LIN {X 0,Y 446.528,Z 466.485,A -85,B 0,C 180,E1 -8829.056,E2 -8829.056} C_VEL
LIN {X 0,Y 446.523,Z 466.485,A -85,B 0,C 180,E1 -8832.73,E2 -8832.73} C_VEL
LIN {X 0,Y 446.485,Z 466.496,A -85,B 0,C 180,E1 -8836.459,E2 -8836.459} C_VEL
LIN {X 0,Y 446.459,Z 466.494,A -85,B 0,C 180,E1 -8839.304,E2 -8839.304} C_VEL
LIN {X 0,Y 446.408,Z 466.501,A -85,B 0,C 180,E1 -8842.2,E2 -8842.2} C_VEL
LIN {X 0,Y 446.448,Z 466.494,A -85,B 0,C 180,E1 -8845.153,E2 -8845.153} C_VEL
LIN {X 0,Y 446.475,Z 466.494,A -85,B 0,C 180,E1 -8848.18,E2 -8848.18} C_VEL
LIN {X 0,Y 446.422,Z 466.498,A -85,B 0,C 180,E1 -8851.3,E2 -8851.3} C_VEL
LIN {X 0,Y 446.423,Z 466.501,A -85,B 0,C 180,E1 -8854.524,E2 -8854.524} C_VEL
LIN {X 0,Y 446.431,Z 466.498,A -85,B 0,C 180,E1 -8858.084,E2 -8858.084} C_VEL
LIN {X 0,Y 446.436,Z 466.501,A -85,B 0,C 180,E1 -8860.921,E2 -8860.921} C_VEL
LIN {X 0,Y 446.395,Z 466.503,A -85,B 0,C 180,E1 -8863.847,E2 -8863.847} C_VEL
LIN {X 0,Y 446.441,Z 466.501,A -85,B 0,C 180,E1 -8866.398,E2 -8866.398} C_VEL
LIN {X 0,Y 446.464,Z 466.495,A -85,B 0,C 180,E1 -8869.806,E2 -8869.806} C_VEL
LIN {X 0,Y 446.43,Z 466.501,A -85,B 0,C 180,E1 -8872.125,E2 -8872.125} C_VEL
LIN {X 0,Y 446.427,Z 466.499,A -85,B 0,C 180,E1 -8875.479,E2 -8875.479} C_VEL
LIN {X 0,Y 446.417,Z 466.5,A -85,B 0,C 180,E1 -8878.701,E2 -8878.701} C_VEL
LIN {X 0,Y 446.482,Z 466.498,A -85,B 0,C 180,E1 -8881.823,E2 -8881.823} C_VEL
LIN {X 0,Y 446.513,Z 466.543,A -85,B 0,C 180,E1 -8882.399,E2 -8882.399} C_VEL
LIN {X 0,Y 449.219,Z 479.048,A -85,B 0,C 180,E1 -8885.015,E2 -8885.015} C_VEL
LIN {X 0,Y 450.113,Z 484.167,A -85,B 0,C 180,E1 -8886.05,E2 -8886.05} C_VEL
LIN {X 0,Y 449.1,Z 500.867,A -85,B 0,C 180,E1 -8889.146,E2 -8889.146} C_VEL
LIN {X 0,Y 448.277,Z 515.978,A -85,B 0,C 180,E1 -8891.866,E2 -8891.866} C_VEL
LIN {X 0,Y 451.84,Z 534.729,A -85,B 0,C 180,E1 -8892.318,E2 -8892.318} C_VEL
LIN {X 0,Y 451.426,Z 605.013,A -85,B 0,C 180,E1 -8893.355,E2 -8893.355} C_VEL
LIN {X 0,Y 450.704,Z 610.873,A -85,B 0,C 180,E1 -8893.408,E2 -8893.408} C_VEL
LIN {X 0,Y 444.994,Z 629.85,A -85,B 0,C 180,E1 -8893.497,E2 -8893.497} C_VEL
LIN {X 0,Y 444.271,Z 635.605,A -85,B 0,C 180,E1 -8893.63,E2 -8893.63} C_VEL
LIN {X 0,Y 443.946,Z 647.952,A -85,B 0,C 180,E1 -8894.095,E2 -8894.095} C_VEL
LIN {X 0,Y 443.491,Z 657.945,A -85,B 0,C 180,E1 -8894.608,E2 -8894.608} C_VEL
LIN {X 0,Y 442.878,Z 668.385,A -85,B 0,C 180,E1 -8895.293,E2 -8895.293} C_VEL
LIN {X 0,Y 442.237,Z 679.403,A -85,B 0,C 180,E1 -8896.21,E2 -8896.21} C_VEL
LIN {X 0,Y 441.507,Z 688.316,A -85,B 0,C 180,E1 -8897.125,E2 -8897.125} C_VEL
LIN {X 0,Y 440.928,Z 697.479,A -85,B 0,C 180,E1 -8898.276,E2 -8898.276} C_VEL
LIN {X 0,Y 440.202,Z 706.324,A -85,B 0,C 180,E1 -8899.654,E2 -8899.654} C_VEL
LIN {X 0,Y 439.593,Z 713.46,A -85,B 0,C 180,E1 -8901.034,E2 -8901.034} C_VEL
LIN {X 0,Y 439.08,Z 720.054,A -85,B 0,C 180,E1 -8902.644,E2 -8902.644} C_VEL
LIN {X 0,Y 438.785,Z 724.416,A -85,B 0,C 180,E1 -8904.025,E2 -8904.025} C_VEL
LIN {X 0,Y 438.668,Z 727.741,A -85,B 0,C 180,E1 -8905.407,E2 -8905.407} C_VEL
LIN {X 0,Y 438.601,Z 729.446,A -85,B 0,C 180,E1 -8906.326,E2 -8906.326} C_VEL
LIN {X 0,Y 438.436,Z 731.666,A -85,B 0,C 180,E1 -8908.164,E2 -8908.164} C_VEL
LIN {X 0,Y 438.341,Z 732.451,A -85,B 0,C 180,E1 -8910.001,E2 -8910.001} C_VEL
LIN {X 0,Y 438.436,Z 731.738,A -85,B 0,C 180,E1 -8911.838,E2 -8911.838} C_VEL
LIN {X 0,Y 438.589,Z 729.577,A -85,B 0,C 180,E1 -8913.676,E2 -8913.676} C_VEL
LIN {X 0,Y 438.611,Z 726.93,A -85,B 0,C 180,E1 -8915.057,E2 -8915.057} C_VEL
LIN {X 0,Y 438.945,Z 723.319,A -85,B 0,C 180,E1 -8916.436,E2 -8916.436} C_VEL
LIN {X 0,Y 439.215,Z 718.662,A -85,B 0,C 180,E1 -8917.818,E2 -8917.818} C_VEL
LIN {X 0,Y 439.685,Z 712.8,A -85,B 0,C 180,E1 -8919.199,E2 -8919.199} C_VEL
LIN {X 0,Y 440.228,Z 705.527,A -85,B 0,C 180,E1 -8920.58,E2 -8920.58} C_VEL
LIN {X 0,Y 440.799,Z 698.102,A -85,B 0,C 180,E1 -8921.73,E2 -8921.73} C_VEL
LIN {X 0,Y 441.496,Z 689.112,A -85,B 0,C 180,E1 -8922.878,E2 -8922.878} C_VEL
LIN {X 0,Y 442.302,Z 678.809,A -85,B 0,C 180,E1 -8923.935,E2 -8923.935} C_VEL
LIN {X 0,Y 442.898,Z 668.024,A -85,B 0,C 180,E1 -8924.827,E2 -8924.827} C_VEL
LIN {X 0,Y 443.612,Z 655.51,A -85,B 0,C 180,E1 -8925.625,E2 -8925.625} C_VEL
LIN {X 0,Y 444.08,Z 643.304,A -85,B 0,C 180,E1 -8926.198,E2 -8926.198} C_VEL
LIN {X 0,Y 444.444,Z 630.676,A -85,B 0,C 180,E1 -8926.597,E2 -8926.597} C_VEL
LIN {X 0,Y 444.648,Z 612.531,A -85,B 0,C 180,E1 -8926.914,E2 -8926.914} C_VEL
LIN {X 0,Y 445.096,Z 535.017,A -85,B 0,C 180,E1 -8928.073,E2 -8928.073} C_VEL
LIN {X 0,Y 441.416,Z 515.921,A -85,B 0,C 180,E1 -8928.569,E2 -8928.569} C_VEL
LIN {X 0,Y 442.438,Z 498.957,A -85,B 0,C 180,E1 -8931.675,E2 -8931.675} C_VEL
LIN {X 0,Y 443.258,Z 486.092,A -85,B 0,C 180,E1 -8934.098,E2 -8934.098} C_VEL
LIN {X 0,Y 441.633,Z 477.096,A -85,B 0,C 180,E1 -8935.954,E2 -8935.954} C_VEL
LIN {X 0,Y 439.465,Z 467.377,A -85,B 0,C 180,E1 -8938.046,E2 -8938.046} C_VEL
LIN {X 0,Y 439.367,Z 467.386,A -85,B 0,C 180,E1 -8940.789,E2 -8940.789} C_VEL
LIN {X 0,Y 439.393,Z 467.377,A -85,B 0,C 180,E1 -8944.044,E2 -8944.044} C_VEL
LIN {X 0,Y 439.366,Z 467.383,A -85,B 0,C 180,E1 -8947.435,E2 -8947.435} C_VEL
LIN {X 0,Y 439.42,Z 467.377,A -85,B 0,C 180,E1 -8949.851,E2 -8949.851} C_VEL
LIN {X 0,Y 439.392,Z 467.376,A -85,B 0,C 180,E1 -8952.628,E2 -8952.628} C_VEL
LIN {X 0,Y 439.408,Z 467.372,A -85,B 0,C 180,E1 -8955.271,E2 -8955.271} C_VEL
LIN {X 0,Y 439.394,Z 467.372,A -85,B 0,C 180,E1 -8958.744,E2 -8958.744} C_VEL
LIN {X 0,Y 439.386,Z 467.374,A -85,B 0,C 180,E1 -8961.607,E2 -8961.607} C_VEL
LIN {X 0,Y 439.407,Z 467.372,A -85,B 0,C 180,E1 -8964.844,E2 -8964.844} C_VEL
LIN {X 0,Y 439.379,Z 467.379,A -85,B 0,C 180,E1 -8968.14,E2 -8968.14} C_VEL
LIN {X 0,Y 439.439,Z 467.373,A -85,B 0,C 180,E1 -8971.598,E2 -8971.598} C_VEL
LIN {X 0,Y 439.469,Z 467.447,A -85,B 0,C 180,E1 -8972.222,E2 -8972.222} C_VEL
LIN {X 0,Y 442.662,Z 482.424,A -85,B 0,C 180,E1 -8974.821,E2 -8974.821} C_VEL
LIN {X 0,Y 442.958,Z 486.098,A -85,B 0,C 180,E1 -8975.424,E2 -8975.424} C_VEL
LIN {X 0,Y 442.188,Z 505.789,A -85,B 0,C 180,E1 -8978.558,E2 -8978.558} C_VEL
LIN {X 0,Y 441.378,Z 528.036,A -85,B 0,C 180,E1 -8982.091,E2 -8982.091} C_VEL
LIN {X 0,Y 443.918,Z 544.485,A -85,B 0,C 180,E1 -8982.514,E2 -8982.514} C_VEL
LIN {X 0,Y 442.535,Z 638.568,A -85,B 0,C 180,E1 -8984.278,E2 -8984.278} C_VEL
LIN {X 0,Y 442.265,Z 651.117,A -85,B 0,C 180,E1 -8984.681,E2 -8984.681} C_VEL
LIN {X 0,Y 441.802,Z 664.471,A -85,B 0,C 180,E1 -8985.313,E2 -8985.313} C_VEL
LIN {X 0,Y 441.347,Z 676.321,A -85,B 0,C 180,E1 -8986.063,E2 -8986.063} C_VEL
LIN {X 0,Y 440.881,Z 687.275,A -85,B 0,C 180,E1 -8986.953,E2 -8986.953} C_VEL
LIN {X 0,Y 440.293,Z 697.9,A -85,B 0,C 180,E1 -8988.024,E2 -8988.024} C_VEL
LIN {X 0,Y 439.833,Z 707.197,A -85,B 0,C 180,E1 -8989.178,E2 -8989.178} C_VEL
LIN {X 0,Y 439.374,Z 716.17,A -85,B 0,C 180,E1 -8990.563,E2 -8990.563} C_VEL
LIN {X 0,Y 438.988,Z 723.4,A -85,B 0,C 180,E1 -8991.947,E2 -8991.947} C_VEL
LIN {X 0,Y 438.731,Z 729.051,A -85,B 0,C 180,E1 -8993.307,E2 -8993.307} C_VEL
LIN {X 0,Y 438.605,Z 732.967,A -85,B 0,C 180,E1 -8994.483,E2 -8994.483} C_VEL
LIN {X 0,Y 438.485,Z 736.528,A -85,B 0,C 180,E1 -8995.864,E2 -8995.864} C_VEL
LIN {X 0,Y 438.428,Z 739.05,A -85,B 0,C 180,E1 -8997.243,E2 -8997.243} C_VEL
LIN {X 0,Y 438.35,Z 740.174,A -85,B 0,C 180,E1 -8998.162,E2 -8998.162} C_VEL
LIN {X 0,Y 438.309,Z 740.884,A -85,B 0,C 180,E1 -8999.081,E2 -8999.081} C_VEL
LIN {X 0,Y 438.309,Z 741.198,A -85,B 0,C 180,E1 -9000,E2 -9000} C_VEL
LIN {X 0,Y 438.338,Z 741.073,A -85,B 0,C 180,E1 -9000.919,E2 -9000.919} C_VEL
LIN {X 0,Y 438.374,Z 740.513,A -85,B 0,C 180,E1 -9001.837,E2 -9001.837} C_VEL
LIN {X 0,Y 438.437,Z 739.553,A -85,B 0,C 180,E1 -9002.756,E2 -9002.756} C_VEL
LIN {X 0,Y 438.539,Z 738.167,A -85,B 0,C 180,E1 -9003.675,E2 -9003.675} C_VEL
LIN {X 0,Y 438.517,Z 735.243,A -85,B 0,C 180,E1 -9005.057,E2 -9005.057} C_VEL
LIN {X 0,Y 438.849,Z 731.225,A -85,B 0,C 180,E1 -9006.436,E2 -9006.436} C_VEL
LIN {X 0,Y 439.052,Z 725.028,A -85,B 0,C 180,E1 -9008.051,E2 -9008.051} C_VEL
LIN {X 0,Y 439.494,Z 718.222,A -85,B 0,C 180,E1 -9009.434,E2 -9009.434} C_VEL
LIN {X 0,Y 439.938,Z 709.665,A -85,B 0,C 180,E1 -9010.819,E2 -9010.819} C_VEL
LIN {X 0,Y 440.406,Z 700.881,A -85,B 0,C 180,E1 -9011.973,E2 -9011.973} C_VEL
LIN {X 0,Y 441.01,Z 690.712,A -85,B 0,C 180,E1 -9013.057,E2 -9013.057} C_VEL
LIN {X 0,Y 441.586,Z 679.066,A -85,B 0,C 180,E1 -9014.046,E2 -9014.046} C_VEL
LIN {X 0,Y 442.042,Z 666.93,A -85,B 0,C 180,E1 -9014.855,E2 -9014.855} C_VEL
LIN {X 0,Y 442.577,Z 654.201,A -85,B 0,C 180,E1 -9015.484,E2 -9015.484} C_VEL
LIN {X 0,Y 442.922,Z 642.024,A -85,B 0,C 180,E1 -9015.915,E2 -9015.915} C_VEL
LIN {X 0,Y 443.322,Z 620.082,A -85,B 0,C 180,E1 -9016.373,E2 -9016.373} C_VEL
LIN {X 0,Y 444.614,Z 543.316,A -85,B 0,C 180,E1 -9017.924,E2 -9017.924} C_VEL
LIN {X 0,Y 442.206,Z 530.197,A -85,B 0,C 180,E1 -9018.355,E2 -9018.355} C_VEL
LIN {X 0,Y 442.954,Z 509.029,A -85,B 0,C 180,E1 -9021.647,E2 -9021.647} C_VEL
LIN {X 0,Y 443.703,Z 490.09,A -85,B 0,C 180,E1 -9024.569,E2 -9024.569} C_VEL
LIN {X 0,Y 443.55,Z 484.614,A -85,B 0,C 180,E1 -9025.422,E2 -9025.422} C_VEL
LIN {X 0,Y 441.677,Z 475.467,A -85,B 0,C 180,E1 -9026.99,E2 -9026.99} C_VEL
LIN {X 0,Y 439.434,Z 467.377,A -85,B 0,C 180,E1 -9028.442,E2 -9028.442} C_VEL
LIN {X 0,Y 439.375,Z 467.384,A -85,B 0,C 180,E1 -9032.03,E2 -9032.03} C_VEL
LIN {X 0,Y 439.401,Z 467.377,A -85,B 0,C 180,E1 -9035.34,E2 -9035.34} C_VEL
LIN {X 0,Y 439.395,Z 467.376,A -85,B 0,C 180,E1 -9038.594,E2 -9038.594} C_VEL
LIN {X 0,Y 439.393,Z 467.378,A -85,B 0,C 180,E1 -9041.256,E2 -9041.256} C_VEL
LIN {X 0,Y 439.404,Z 467.375,A -85,B 0,C 180,E1 -9044.729,E2 -9044.729} C_VEL
LIN {X 0,Y 439.4,Z 467.378,A -85,B 0,C 180,E1 -9047.795,E2 -9047.795} C_VEL
LIN {X 0,Y 439.399,Z 467.374,A -85,B 0,C 180,E1 -9050.223,E2 -9050.223} C_VEL
LIN {X 0,Y 439.378,Z 467.38,A -85,B 0,C 180,E1 -9053.712,E2 -9053.712} C_VEL
LIN {X 0,Y 439.377,Z 467.381,A -85,B 0,C 180,E1 -9057.053,E2 -9057.053} C_VEL
LIN {X 0,Y 439.4,Z 467.425,A -85,B 0,C 180,E1 -9059.823,E2 -9059.823} C_VEL
LIN {X 0,Y 443.454,Z 483.224,A -85,B 0,C 180,E1 -9062.561,E2 -9062.561} C_VEL
LIN {X 0,Y 445.005,Z 490.464,A -85,B 0,C 180,E1 -9063.754,E2 -9063.754} C_VEL
LIN {X 0,Y 443.575,Z 510.491,A -85,B 0,C 180,E1 -9066.664,E2 -9066.664} C_VEL
LIN {X 0,Y 442.748,Z 522.844,A -85,B 0,C 180,E1 -9068.447,E2 -9068.447} C_VEL
LIN {X 0,Y 445.963,Z 544.781,A -85,B 0,C 180,E1 -9068.984,E2 -9068.984} C_VEL
LIN {X 0,Y 444.312,Z 657.862,A -85,B 0,C 180,E1 -9070.958,E2 -9070.958} C_VEL
LIN {X 0,Y 443.803,Z 672.315,A -85,B 0,C 180,E1 -9071.385,E2 -9071.385} C_VEL
LIN {X 0,Y 443.198,Z 685.875,A -85,B 0,C 180,E1 -9071.966,E2 -9071.966} C_VEL
LIN {X 0,Y 442.454,Z 700.183,A -85,B 0,C 180,E1 -9072.791,E2 -9072.791} C_VEL
LIN {X 0,Y 441.713,Z 712.707,A -85,B 0,C 180,E1 -9073.713,E2 -9073.713} C_VEL
LIN {X 0,Y 440.951,Z 724.181,A -85,B 0,C 180,E1 -9074.752,E2 -9074.752} C_VEL
LIN {X 0,Y 440.283,Z 734.747,A -85,B 0,C 180,E1 -9075.91,E2 -9075.91} C_VEL
LIN {X 0,Y 439.755,Z 744.042,A -85,B 0,C 180,E1 -9077.13,E2 -9077.13} C_VEL
LIN {X 0,Y 439.299,Z 752.571,A -85,B 0,C 180,E1 -9078.463,E2 -9078.463} C_VEL
LIN {X 0,Y 438.854,Z 761.143,A -85,B 0,C 180,E1 -9080.086,E2 -9080.086} C_VEL
LIN {X 0,Y 438.578,Z 768.005,A -85,B 0,C 180,E1 -9081.707,E2 -9081.707} C_VEL
LIN {X 0,Y 438.46,Z 772.747,A -85,B 0,C 180,E1 -9083.094,E2 -9083.094} C_VEL
LIN {X 0,Y 438.417,Z 777.575,A -85,B 0,C 180,E1 -9084.941,E2 -9084.941} C_VEL
LIN {X 0,Y 438.347,Z 780.144,A -85,B 0,C 180,E1 -9086.322,E2 -9086.322} C_VEL
LIN {X 0,Y 438.407,Z 781.414,A -85,B 0,C 180,E1 -9087.242,E2 -9087.242} C_VEL
LIN {X 0,Y 438.364,Z 782.86,A -85,B 0,C 180,E1 -9089.08,E2 -9089.08} C_VEL
LIN {X 0,Y 438.363,Z 782.861,A -85,B 0,C 180,E1 -9090.917,E2 -9090.917} C_VEL
LIN {X 0,Y 438.406,Z 781.418,A -85,B 0,C 180,E1 -9092.755,E2 -9092.755} C_VEL
LIN {X 0,Y 438.35,Z 778.515,A -85,B 0,C 180,E1 -9094.597,E2 -9094.597} C_VEL
LIN {X 0,Y 438.442,Z 774.291,A -85,B 0,C 180,E1 -9096.369,E2 -9096.369} C_VEL
LIN {X 0,Y 438.502,Z 769.686,A -85,B 0,C 180,E1 -9097.829,E2 -9097.829} C_VEL
LIN {X 0,Y 438.776,Z 763.241,A -85,B 0,C 180,E1 -9099.448,E2 -9099.448} C_VEL
LIN {X 0,Y 439.159,Z 755.192,A -85,B 0,C 180,E1 -9101.071,E2 -9101.071} C_VEL
LIN {X 0,Y 439.54,Z 747.348,A -85,B 0,C 180,E1 -9102.376,E2 -9102.376} C_VEL
LIN {X 0,Y 440.193,Z 736.626,A -85,B 0,C 180,E1 -9103.855,E2 -9103.855} C_VEL
LIN {X 0,Y 440.921,Z 725.347,A -85,B 0,C 180,E1 -9105.128,E2 -9105.128} C_VEL
LIN {X 0,Y 441.654,Z 714.136,A -85,B 0,C 180,E1 -9106.168,E2 -9106.168} C_VEL
LIN {X 0,Y 442.323,Z 701.958,A -85,B 0,C 180,E1 -9107.093,E2 -9107.093} C_VEL
LIN {X 0,Y 443.048,Z 689.083,A -85,B 0,C 180,E1 -9107.867,E2 -9107.867} C_VEL
LIN {X 0,Y 443.667,Z 675.303,A -85,B 0,C 180,E1 -9108.499,E2 -9108.499} C_VEL
LIN {X 0,Y 444.218,Z 661.187,A -85,B 0,C 180,E1 -9108.954,E2 -9108.954} C_VEL
LIN {X 0,Y 444.603,Z 640.583,A -85,B 0,C 180,E1 -9109.356,E2 -9109.356} C_VEL
LIN {X 0,Y 445.85,Z 543.854,A -85,B 0,C 180,E1 -9111.033,E2 -9111.033} C_VEL
LIN {X 0,Y 442.72,Z 522.592,A -85,B 0,C 180,E1 -9111.566,E2 -9111.566} C_VEL
LIN {X 0,Y 444.176,Z 502.158,A -85,B 0,C 180,E1 -9114.539,E2 -9114.539} C_VEL
LIN {X 0,Y 444.99,Z 490.428,A -85,B 0,C 180,E1 -9116.244,E2 -9116.244} C_VEL
LIN {X 0,Y 441.733,Z 476.236,A -85,B 0,C 180,E1 -9118.621,E2 -9118.621} C_VEL
LIN {X 0,Y 439.4,Z 467.374,A -85,B 0,C 180,E1 -9120.177,E2 -9120.177} C_VEL
LIN {X 0,Y 439.391,Z 467.374,A -85,B 0,C 180,E1 -9123.723,E2 -9123.723} C_VEL
LIN {X 0,Y 439.353,Z 467.384,A -85,B 0,C 180,E1 -9126.888,E2 -9126.888} C_VEL
LIN {X 0,Y 439.422,Z 467.372,A -85,B 0,C 180,E1 -9129.852,E2 -9129.852} C_VEL
LIN {X 0,Y 439.396,Z 467.379,A -85,B 0,C 180,E1 -9132.629,E2 -9132.629} C_VEL
LIN {X 0,Y 439.395,Z 467.373,A -85,B 0,C 180,E1 -9136.032,E2 -9136.032} C_VEL
LIN {X 0,Y 439.392,Z 467.375,A -85,B 0,C 180,E1 -9139.021,E2 -9139.021} C_VEL
LIN {X 0,Y 439.384,Z 467.372,A -85,B 0,C 180,E1 -9141.604,E2 -9141.604} C_VEL
LIN {X 0,Y 439.391,Z 467.365,A -85,B 0,C 180,E1 -9144.843,E2 -9144.843} C_VEL
LIN {X 0,Y 439.378,Z 467.376,A -85,B 0,C 180,E1 -9148.14,E2 -9148.14} C_VEL
LIN {X 0,Y 439.415,Z 467.37,A -85,B 0,C 180,E1 -9151.326,E2 -9151.326} C_VEL
LIN {X 0,Y 439.395,Z 467.379,A -85,B 0,C 180,E1 -9154.415,E2 -9154.415} C_VEL
LIN {X 0,Y 439.354,Z 467.361,A -85,B 0,C 180,E1 -9157.424,E2 -9157.424} C_VEL
LIN {X 0,Y 439.43,Z 467.37,A -85,B 0,C 180,E1 -9160.662,E2 -9160.662} C_VEL
LIN {X 0,Y 439.451,Z 467.366,A -85,B 0,C 180,E1 -9164.224,E2 -9164.224} C_VEL
LIN {X 0,Y 439.501,Z 467.36,A -85,B 0,C 180,E1 -9168.002,E2 -9168.002} C_VEL
LIN {X 0,Y 439.536,Z 467.356,A -85,B 0,C 180,E1 -9171.726,E2 -9171.726} C_VEL
LIN {X 0,Y 439.614,Z 467.346,A -85,B 0,C 180,E1 -9174.496,E2 -9174.496} C_VEL
LIN {X 0,Y 439.626,Z 467.345,A -85,B 0,C 180,E1 -9178.168,E2 -9178.168} C_VEL
LIN {X 0,Y 439.754,Z 467.328,A -85,B 0,C 180,E1 -9180,E2 -9180} C_VEL
LIN {X 0,Y 439.646,Z 467.34,A -85,B 0,C 180,E1 -9182.749,E2 -9182.749} C_VEL
LIN {X 0,Y 439.607,Z 467.353,A -85,B 0,C 180,E1 -9186.426,E2 -9186.426} C_VEL
LIN {X 0,Y 439.491,Z 467.36,A -85,B 0,C 180,E1 -9189.202,E2 -9189.202} C_VEL
LIN {X 0,Y 439.493,Z 467.36,A -85,B 0,C 180,E1 -9192.727,E2 -9192.727} C_VEL
LIN {X 0,Y 439.449,Z 467.372,A -85,B 0,C 180,E1 -9196.355,E2 -9196.355} C_VEL
LIN {X 0,Y 439.392,Z 467.374,A -85,B 0,C 180,E1 -9199.627,E2 -9199.627} C_VEL
LIN {X 0,Y 439.355,Z 467.38,A -85,B 0,C 180,E1 -9202.576,E2 -9202.576} C_VEL
LIN {X 0,Y 439.395,Z 467.372,A -85,B 0,C 180,E1 -9205.586,E2 -9205.586} C_VEL
LIN {X 0,Y 439.416,Z 467.375,A -85,B 0,C 180,E1 -9208.674,E2 -9208.674} C_VEL
LIN {X 0,Y 439.376,Z 467.378,A -85,B 0,C 180,E1 -9212.035,E2 -9212.035} C_VEL
LIN {X 0,Y 439.388,Z 467.375,A -85,B 0,C 180,E1 -9215.342,E2 -9215.342} C_VEL
LIN {X 0,Y 439.392,Z 467.381,A -85,B 0,C 180,E1 -9218.594,E2 -9218.594} C_VEL
LIN {X 0,Y 439.391,Z 467.376,A -85,B 0,C 180,E1 -9221.26,E2 -9221.26} C_VEL
LIN {X 0,Y 439.396,Z 467.378,A -85,B 0,C 180,E1 -9224.73,E2 -9224.73} C_VEL
LIN {X 0,Y 439.407,Z 467.374,A -85,B 0,C 180,E1 -9227.799,E2 -9227.799} C_VEL
LIN {X 0,Y 439.447,Z 467.371,A -85,B 0,C 180,E1 -9230.232,E2 -9230.232} C_VEL
LIN {X 0,Y 439.373,Z 467.374,A -85,B 0,C 180,E1 -9233.715,E2 -9233.715} C_VEL
LIN {X 0,Y 439.372,Z 467.381,A -85,B 0,C 180,E1 -9237.056,E2 -9237.056} C_VEL
LIN {X 0,Y 439.394,Z 467.378,A -85,B 0,C 180,E1 -9240.277,E2 -9240.277} C_VEL
LIN {X 0,Y 439.47,Z 467.469,A -85,B 0,C 180,E1 -9242.075,E2 -9242.075} C_VEL
LIN {X 0,Y 442.059,Z 479.194,A -85,B 0,C 180,E1 -9244.581,E2 -9244.581} C_VEL
LIN {X 0,Y 443.239,Z 485.599,A -85,B 0,C 180,E1 -9245.904,E2 -9245.904} C_VEL
LIN {X 0,Y 442.203,Z 502.354,A -85,B 0,C 180,E1 -9249.049,E2 -9249.049} C_VEL
LIN {X 0,Y 441.418,Z 515.939,A -85,B 0,C 180,E1 -9251.529,E2 -9251.529} C_VEL
LIN {X 0,Y 445.158,Z 535.672,A -85,B 0,C 180,E1 -9252.031,E2 -9252.031} C_VEL
LIN {X 0,Y 444.466,Z 628.207,A -85,B 0,C 180,E1 -9253.436,E2 -9253.436} C_VEL
LIN {X 0,Y 444.271,Z 635.605,A -85,B 0,C 180,E1 -9253.63,E2 -9253.63} C_VEL
LIN {X 0,Y 443.847,Z 639.428,A -85,B 0,C 180,E1 -9253.738,E2 -9253.738} C_VEL
LIN {X 0,Y 441.761,Z 646.881,A -85,B 0,C 180,E1 -9253.951,E2 -9253.951} C_VEL
LIN {X 0,Y 437.525,Z 658.588,A -85,B 0,C 180,E1 -9254.396,E2 -9254.396} C_VEL
LIN {X 0,Y 436.357,Z 664.758,A -85,B 0,C 180,E1 -9254.754,E2 -9254.754} C_VEL
LIN {X 0,Y 435.632,Z 676.154,A -85,B 0,C 180,E1 -9255.64,E2 -9255.64} C_VEL
LIN {X 0,Y 434.826,Z 686.741,A -85,B 0,C 180,E1 -9256.685,E2 -9256.685} C_VEL
LIN {X 0,Y 434.119,Z 696.253,A -85,B 0,C 180,E1 -9257.852,E2 -9257.852} C_VEL
LIN {X 0,Y 433.437,Z 704.057,A -85,B 0,C 180,E1 -9259.018,E2 -9259.018} C_VEL
LIN {X 0,Y 432.835,Z 711.727,A -85,B 0,C 180,E1 -9260.421,E2 -9260.421} C_VEL
LIN {X 0,Y 432.35,Z 716.928,A -85,B 0,C 180,E1 -9261.589,E2 -9261.589} C_VEL
LIN {X 0,Y 431.954,Z 721.974,A -85,B 0,C 180,E1 -9262.974,E2 -9262.974} C_VEL
LIN {X 0,Y 431.603,Z 726.039,A -85,B 0,C 180,E1 -9264.394,E2 -9264.394} C_VEL
LIN {X 0,Y 431.587,Z 728.162,A -85,B 0,C 180,E1 -9265.331,E2 -9265.331} C_VEL
LIN {X 0,Y 431.544,Z 729.86,A -85,B 0,C 180,E1 -9266.266,E2 -9266.266} C_VEL
LIN {X 0,Y 431.353,Z 732.076,A -85,B 0,C 180,E1 -9268.134,E2 -9268.134} C_VEL
LIN {X 0,Y 431.281,Z 732.859,A -85,B 0,C 180,E1 -9270.001,E2 -9270.001} C_VEL
LIN {X 0,Y 431.353,Z 732.148,A -85,B 0,C 180,E1 -9271.869,E2 -9271.869} C_VEL
LIN {X 0,Y 431.533,Z 729.989,A -85,B 0,C 180,E1 -9273.736,E2 -9273.736} C_VEL
LIN {X 0,Y 431.539,Z 727.349,A -85,B 0,C 180,E1 -9275.14,E2 -9275.14} C_VEL
LIN {X 0,Y 431.91,Z 723.744,A -85,B 0,C 180,E1 -9276.542,E2 -9276.542} C_VEL
LIN {X 0,Y 432.181,Z 719.097,A -85,B 0,C 180,E1 -9277.946,E2 -9277.946} C_VEL
LIN {X 0,Y 432.699,Z 713.245,A -85,B 0,C 180,E1 -9279.349,E2 -9279.349} C_VEL
LIN {X 0,Y 433.282,Z 705.984,A -85,B 0,C 180,E1 -9280.752,E2 -9280.752} C_VEL
LIN {X 0,Y 433.872,Z 698.578,A -85,B 0,C 180,E1 -9281.92,E2 -9281.92} C_VEL
LIN {X 0,Y 434.614,Z 689.615,A -85,B 0,C 180,E1 -9283.086,E2 -9283.086} C_VEL
LIN {X 0,Y 435.432,Z 679.539,A -85,B 0,C 180,E1 -9284.142,E2 -9284.142} C_VEL
LIN {X 0,Y 436.068,Z 668.622,A -85,B 0,C 180,E1 -9285.064,E2 -9285.064} C_VEL
LIN {X 0,Y 436.806,Z 656.18,A -85,B 0,C 180,E1 -9285.875,E2 -9285.875} C_VEL
LIN {X 0,Y 437.336,Z 643.401,A -85,B 0,C 180,E1 -9286.484,E2 -9286.484} C_VEL
LIN {X 0,Y 437.737,Z 630.664,A -85,B 0,C 180,E1 -9286.889,E2 -9286.889} C_VEL
LIN {X 0,Y 437.945,Z 612.328,A -85,B 0,C 180,E1 -9287.211,E2 -9287.211} C_VEL
LIN {X 0,Y 438.491,Z 536.306,A -85,B 0,C 180,E1 -9288.362,E2 -9288.362} C_VEL
LIN {X 0,Y 434.59,Z 515.966,A -85,B 0,C 180,E1 -9288.902,E2 -9288.902} C_VEL
LIN {X 0,Y 435.698,Z 497.838,A -85,B 0,C 180,E1 -9292.277,E2 -9292.277} C_VEL
LIN {X 0,Y 436.402,Z 487.52,A -85,B 0,C 180,E1 -9294.248,E2 -9294.248} C_VEL
LIN {X 0,Y 434.447,Z 477.241,A -85,B 0,C 180,E1 -9296.416,E2 -9296.416} C_VEL
LIN {X 0,Y 432.401,Z 468.255,A -85,B 0,C 180,E1 -9298.426,E2 -9298.426} C_VEL
LIN {X 0,Y 432.327,Z 468.262,A -85,B 0,C 180,E1 -9301.347,E2 -9301.347} C_VEL
LIN {X 0,Y 432.346,Z 468.253,A -85,B 0,C 180,E1 -9304.678,E2 -9304.678} C_VEL
LIN {X 0,Y 432.353,Z 468.251,A -85,B 0,C 180,E1 -9308.149,E2 -9308.149} C_VEL
LIN {X 0,Y 432.341,Z 468.255,A -85,B 0,C 180,E1 -9311.603,E2 -9311.603} C_VEL
LIN {X 0,Y 432.347,Z 468.25,A -85,B 0,C 180,E1 -9314.347,E2 -9314.347} C_VEL
LIN {X 0,Y 432.326,Z 468.255,A -85,B 0,C 180,E1 -9317.016,E2 -9317.016} C_VEL
LIN {X 0,Y 432.34,Z 468.258,A -85,B 0,C 180,E1 -9319.821,E2 -9319.821} C_VEL
LIN {X 0,Y 432.321,Z 468.251,A -85,B 0,C 180,E1 -9323.023,E2 -9323.023} C_VEL
LIN {X 0,Y 432.366,Z 468.254,A -85,B 0,C 180,E1 -9325.997,E2 -9325.997} C_VEL
LIN {X 0,Y 432.353,Z 468.257,A -85,B 0,C 180,E1 -9329.49,E2 -9329.49} C_VEL
LIN {X 0,Y 432.437,Z 468.307,A -85,B 0,C 180,E1 -9331.979,E2 -9331.979} C_VEL
LIN {X 0,Y 435.842,Z 484.382,A -85,B 0,C 180,E1 -9334.782,E2 -9334.782} C_VEL
LIN {X 0,Y 436.032,Z 488.571,A -85,B 0,C 180,E1 -9335.478,E2 -9335.478} C_VEL
LIN {X 0,Y 435.149,Z 510.194,A -85,B 0,C 180,E1 -9338.939,E2 -9338.939} C_VEL
LIN {X 0,Y 434.479,Z 528.296,A -85,B 0,C 180,E1 -9341.833,E2 -9341.833} C_VEL
LIN {X 0,Y 437.095,Z 545.583,A -85,B 0,C 180,E1 -9342.285,E2 -9342.285} C_VEL
LIN {X 0,Y 435.645,Z 638.007,A -85,B 0,C 180,E1 -9344.052,E2 -9344.052} C_VEL
LIN {X 0,Y 435.351,Z 651.582,A -85,B 0,C 180,E1 -9344.492,E2 -9344.492} C_VEL
LIN {X 0,Y 434.862,Z 664.878,A -85,B 0,C 180,E1 -9345.134,E2 -9345.134} C_VEL
LIN {X 0,Y 434.351,Z 677.475,A -85,B 0,C 180,E1 -9345.953,E2 -9345.953} C_VEL
LIN {X 0,Y 433.836,Z 688.639,A -85,B 0,C 180,E1 -9346.891,E2 -9346.891} C_VEL
LIN {X 0,Y 433.278,Z 698.797,A -85,B 0,C 180,E1 -9347.945,E2 -9347.945} C_VEL
LIN {X 0,Y 432.831,Z 707.15,A -85,B 0,C 180,E1 -9349.001,E2 -9349.001} C_VEL
LIN {X 0,Y 432.339,Z 716.207,A -85,B 0,C 180,E1 -9350.408,E2 -9350.408} C_VEL
LIN {X 0,Y 431.954,Z 723.5,A -85,B 0,C 180,E1 -9351.815,E2 -9351.815} C_VEL
LIN {X 0,Y 431.659,Z 729.59,A -85,B 0,C 180,E1 -9353.303,E2 -9353.303} C_VEL
LIN {X 0,Y 431.445,Z 734.474,A -85,B 0,C 180,E1 -9354.86,E2 -9354.86} C_VEL
LIN {X 0,Y 431.404,Z 737.715,A -85,B 0,C 180,E1 -9356.264,E2 -9356.264} C_VEL
LIN {X 0,Y 431.36,Z 739.327,A -85,B 0,C 180,E1 -9357.198,E2 -9357.198} C_VEL
LIN {X 0,Y 431.271,Z 740.479,A -85,B 0,C 180,E1 -9358.132,E2 -9358.132} C_VEL
LIN {X 0,Y 431.223,Z 741.205,A -85,B 0,C 180,E1 -9359.066,E2 -9359.066} C_VEL
LIN {X 0,Y 431.221,Z 741.533,A -85,B 0,C 180,E1 -9360,E2 -9360} C_VEL
LIN {X 0,Y 431.251,Z 741.433,A -85,B 0,C 180,E1 -9360.934,E2 -9360.934} C_VEL
LIN {X 0,Y 431.294,Z 740.886,A -85,B 0,C 180,E1 -9361.867,E2 -9361.867} C_VEL
LIN {X 0,Y 431.37,Z 739.939,A -85,B 0,C 180,E1 -9362.801,E2 -9362.801} C_VEL
LIN {X 0,Y 431.48,Z 738.574,A -85,B 0,C 180,E1 -9363.735,E2 -9363.735} C_VEL
LIN {X 0,Y 431.458,Z 735.674,A -85,B 0,C 180,E1 -9365.14,E2 -9365.14} C_VEL
LIN {X 0,Y 431.785,Z 731.671,A -85,B 0,C 180,E1 -9366.542,E2 -9366.542} C_VEL
LIN {X 0,Y 432.045,Z 725.475,A -85,B 0,C 180,E1 -9368.183,E2 -9368.183} C_VEL
LIN {X 0,Y 432.511,Z 718.675,A -85,B 0,C 180,E1 -9369.587,E2 -9369.587} C_VEL
LIN {X 0,Y 432.989,Z 710.118,A -85,B 0,C 180,E1 -9370.995,E2 -9370.995} C_VEL
LIN {X 0,Y 433.479,Z 701.367,A -85,B 0,C 180,E1 -9372.167,E2 -9372.167} C_VEL
LIN {X 0,Y 434.112,Z 691.379,A -85,B 0,C 180,E1 -9373.258,E2 -9373.258} C_VEL
LIN {X 0,Y 434.746,Z 679.724,A -85,B 0,C 180,E1 -9374.272,E2 -9374.272} C_VEL
LIN {X 0,Y 435.244,Z 667.735,A -85,B 0,C 180,E1 -9375.092,E2 -9375.092} C_VEL
LIN {X 0,Y 435.839,Z 653.807,A -85,B 0,C 180,E1 -9375.79,E2 -9375.79} C_VEL
LIN {X 0,Y 436.206,Z 641.176,A -85,B 0,C 180,E1 -9376.226,E2 -9376.226} C_VEL
LIN {X 0,Y 438.103,Z 544.661,A -85,B 0,C 180,E1 -9378.248,E2 -9378.248} C_VEL
LIN {X 0,Y 435.49,Z 530.58,A -85,B 0,C 180,E1 -9378.732,E2 -9378.732} C_VEL
LIN {X 0,Y 436.242,Z 511.407,A -85,B 0,C 180,E1 -9381.749,E2 -9381.749} C_VEL
LIN {X 0,Y 437.099,Z 491.01,A -85,B 0,C 180,E1 -9384.929,E2 -9384.929} C_VEL
LIN {X 0,Y 436.828,Z 485.912,A -85,B 0,C 180,E1 -9385.747,E2 -9385.747} C_VEL
LIN {X 0,Y 434.639,Z 475.975,A -85,B 0,C 180,E1 -9387.498,E2 -9387.498} C_VEL
LIN {X 0,Y 432.355,Z 468.26,A -85,B 0,C 180,E1 -9388.945,E2 -9388.945} C_VEL
LIN {X 0,Y 432.33,Z 468.261,A -85,B 0,C 180,E1 -9392.293,E2 -9392.293} C_VEL
LIN {X 0,Y 432.346,Z 468.256,A -85,B 0,C 180,E1 -9394.676,E2 -9394.676} C_VEL
LIN {X 0,Y 432.352,Z 468.256,A -85,B 0,C 180,E1 -9398.148,E2 -9398.148} C_VEL
LIN {X 0,Y 432.337,Z 468.257,A -85,B 0,C 180,E1 -9401.601,E2 -9401.601} C_VEL
LIN {X 0,Y 432.338,Z 468.257,A -85,B 0,C 180,E1 -9404.347,E2 -9404.347} C_VEL
LIN {X 0,Y 432.324,Z 468.257,A -85,B 0,C 180,E1 -9407.015,E2 -9407.015} C_VEL
LIN {X 0,Y 432.338,Z 468.258,A -85,B 0,C 180,E1 -9409.82,E2 -9409.82} C_VEL
LIN {X 0,Y 432.31,Z 468.258,A -85,B 0,C 180,E1 -9413.021,E2 -9413.021} C_VEL
LIN {X 0,Y 432.364,Z 468.254,A -85,B 0,C 180,E1 -9415.996,E2 -9415.996} C_VEL
LIN {X 0,Y 432.354,Z 468.298,A -85,B 0,C 180,E1 -9419.444,E2 -9419.444} C_VEL
LIN {X 0,Y 436.525,Z 484.488,A -85,B 0,C 180,E1 -9422.312,E2 -9422.312} C_VEL
LIN {X 0,Y 438.132,Z 491.733,A -85,B 0,C 180,E1 -9423.534,E2 -9423.534} C_VEL
LIN {X 0,Y 437.611,Z 500.302,A -85,B 0,C 180,E1 -9424.811,E2 -9424.811} C_VEL
LIN {X 0,Y 435.904,Z 522.612,A -85,B 0,C 180,E1 -9428.108,E2 -9428.108} C_VEL
LIN {X 0,Y 439.23,Z 545.177,A -85,B 0,C 180,E1 -9428.681,E2 -9428.681} C_VEL
LIN {X 0,Y 437.534,Z 657.857,A -85,B 0,C 180,E1 -9430.682,E2 -9430.682} C_VEL
LIN {X 0,Y 437.027,Z 672.201,A -85,B 0,C 180,E1 -9431.116,E2 -9431.116} C_VEL
LIN {X 0,Y 436.414,Z 684.806,A -85,B 0,C 180,E1 -9431.658,E2 -9431.658} C_VEL
LIN {X 0,Y 435.714,Z 697.759,A -85,B 0,C 180,E1 -9432.395,E2 -9432.395} C_VEL
LIN {X 0,Y 434.983,Z 710.677,A -85,B 0,C 180,E1 -9433.333,E2 -9433.333} C_VEL
LIN {X 0,Y 434.121,Z 722.437,A -85,B 0,C 180,E1 -9434.386,E2 -9434.386} C_VEL
LIN {X 0,Y 433.317,Z 734.229,A -85,B 0,C 180,E1 -9435.679,E2 -9435.679} C_VEL
LIN {X 0,Y 432.729,Z 744.293,A -85,B 0,C 180,E1 -9437.025,E2 -9437.025} C_VEL
LIN {X 0,Y 432.216,Z 753.45,A -85,B 0,C 180,E1 -9438.509,E2 -9438.509} C_VEL
LIN {X 0,Y 431.755,Z 761.739,A -85,B 0,C 180,E1 -9440.158,E2 -9440.158} C_VEL
LIN {X 0,Y 431.492,Z 767.565,A -85,B 0,C 180,E1 -9441.57,E2 -9441.57} C_VEL
LIN {X 0,Y 431.373,Z 773.657,A -85,B 0,C 180,E1 -9443.45,E2 -9443.45} C_VEL
LIN {X 0,Y 431.283,Z 778.09,A -85,B 0,C 180,E1 -9445.325,E2 -9445.325} C_VEL
LIN {X 0,Y 431.332,Z 781.002,A -85,B 0,C 180,E1 -9447.197,E2 -9447.197} C_VEL
LIN {X 0,Y 431.274,Z 782.45,A -85,B 0,C 180,E1 -9449.065,E2 -9449.065} C_VEL
LIN {X 0,Y 431.273,Z 782.451,A -85,B 0,C 180,E1 -9450.933,E2 -9450.933} C_VEL
LIN {X 0,Y 431.332,Z 781.006,A -85,B 0,C 180,E1 -9452.801,E2 -9452.801} C_VEL
LIN {X 0,Y 431.282,Z 778.096,A -85,B 0,C 180,E1 -9454.672,E2 -9454.672} C_VEL
LIN {X 0,Y 431.371,Z 773.659,A -85,B 0,C 180,E1 -9456.547,E2 -9456.547} C_VEL
LIN {X 0,Y 431.49,Z 767.565,A -85,B 0,C 180,E1 -9458.428,E2 -9458.428} C_VEL
LIN {X 0,Y 431.781,Z 760.69,A -85,B 0,C 180,E1 -9460.076,E2 -9460.076} C_VEL
LIN {X 0,Y 432.263,Z 752.096,A -85,B 0,C 180,E1 -9461.725,E2 -9461.725} C_VEL
LIN {X 0,Y 432.764,Z 743.116,A -85,B 0,C 180,E1 -9463.14,E2 -9463.14} C_VEL
LIN {X 0,Y 433.453,Z 732.23,A -85,B 0,C 180,E1 -9464.554,E2 -9464.554} C_VEL
LIN {X 0,Y 434.172,Z 721.235,A -85,B 0,C 180,E1 -9465.73,E2 -9465.73} C_VEL
LIN {X 0,Y 435.018,Z 709.224,A -85,B 0,C 180,E1 -9466.784,E2 -9466.784} C_VEL
LIN {X 0,Y 435.803,Z 695.954,A -85,B 0,C 180,E1 -9467.72,E2 -9467.72} C_VEL
LIN {X 0,Y 436.559,Z 681.677,A -85,B 0,C 180,E1 -9468.488,E2 -9468.488} C_VEL
LIN {X 0,Y 437.214,Z 667.074,A -85,B 0,C 180,E1 -9469.056,E2 -9469.056} C_VEL
LIN {X 0,Y 437.698,Z 652.193,A -85,B 0,C 180,E1 -9469.43,E2 -9469.43} C_VEL
LIN {X 0,Y 439.163,Z 544.713,A -85,B 0,C 180,E1 -9471.325,E2 -9471.325} C_VEL
LIN {X 0,Y 435.9,Z 522.551,A -85,B 0,C 180,E1 -9471.89,E2 -9471.89} C_VEL
LIN {X 0,Y 437.463,Z 501.951,A -85,B 0,C 180,E1 -9474.941,E2 -9474.941} C_VEL
LIN {X 0,Y 438.085,Z 491.59,A -85,B 0,C 180,E1 -9476.483,E2 -9476.483} C_VEL
LIN {X 0,Y 435.05,Z 478.478,A -85,B 0,C 180,E1 -9478.723,E2 -9478.723} C_VEL
LIN {X 0,Y 432.345,Z 468.253,A -85,B 0,C 180,E1 -9480.59,E2 -9480.59} C_VEL
LIN {X 0,Y 432.354,Z 468.245,A -85,B 0,C 180,E1 -9484.002,E2 -9484.002} C_VEL
LIN {X 0,Y 432.329,Z 468.258,A -85,B 0,C 180,E1 -9487.198,E2 -9487.198} C_VEL
LIN {X 0,Y 432.352,Z 468.255,A -85,B 0,C 180,E1 -9490.182,E2 -9490.182} C_VEL
LIN {X 0,Y 432.358,Z 468.254,A -85,B 0,C 180,E1 -9493.054,E2 -9493.054} C_VEL
LIN {X 0,Y 432.37,Z 468.247,A -85,B 0,C 180,E1 -9495.657,E2 -9495.657} C_VEL
LIN {X 0,Y 432.365,Z 468.25,A -85,B 0,C 180,E1 -9498.391,E2 -9498.391} C_VEL
LIN {X 0,Y 432.344,Z 468.25,A -85,B 0,C 180,E1 -9501.851,E2 -9501.851} C_VEL
LIN {X 0,Y 432.331,Z 468.248,A -85,B 0,C 180,E1 -9505.322,E2 -9505.322} C_VEL
LIN {X 0,Y 432.323,Z 468.255,A -85,B 0,C 180,E1 -9508.654,E2 -9508.654} C_VEL
LIN {X 0,Y 432.374,Z 468.246,A -85,B 0,C 180,E1 -9511.876,E2 -9511.876} C_VEL
LIN {X 0,Y 432.341,Z 468.252,A -85,B 0,C 180,E1 -9514.998,E2 -9514.998} C_VEL
LIN {X 0,Y 432.346,Z 468.233,A -85,B 0,C 180,E1 -9518.045,E2 -9518.045} C_VEL
LIN {X 0,Y 432.375,Z 468.251,A -85,B 0,C 180,E1 -9521.029,E2 -9521.029} C_VEL
LIN {X 0,Y 432.419,Z 468.24,A -85,B 0,C 180,E1 -9523.961,E2 -9523.961} C_VEL
LIN {X 0,Y 432.472,Z 468.235,A -85,B 0,C 180,E1 -9527.804,E2 -9527.804} C_VEL
LIN {X 0,Y 432.481,Z 468.235,A -85,B 0,C 180,E1 -9531.59,E2 -9531.59} C_VEL
LIN {X 0,Y 432.59,Z 468.219,A -85,B 0,C 180,E1 -9534.406,E2 -9534.406} C_VEL
LIN {X 0,Y 432.595,Z 468.22,A -85,B 0,C 180,E1 -9538.138,E2 -9538.138} C_VEL
LIN {X 0,Y 432.724,Z 468.204,A -85,B 0,C 180,E1 -9540,E2 -9540} C_VEL
LIN {X 0,Y 432.596,Z 468.218,A -85,B 0,C 180,E1 -9542.794,E2 -9542.794} C_VEL
LIN {X 0,Y 432.562,Z 468.231,A -85,B 0,C 180,E1 -9546.531,E2 -9546.531} C_VEL
LIN {X 0,Y 432.434,Z 468.239,A -85,B 0,C 180,E1 -9549.353,E2 -9549.353} C_VEL
LIN {X 0,Y 432.433,Z 468.239,A -85,B 0,C 180,E1 -9552.812,E2 -9552.812} C_VEL
LIN {X 0,Y 432.412,Z 468.248,A -85,B 0,C 180,E1 -9556.484,E2 -9556.484} C_VEL
LIN {X 0,Y 432.329,Z 468.255,A -85,B 0,C 180,E1 -9559.961,E2 -9559.961} C_VEL
LIN {X 0,Y 432.309,Z 468.258,A -85,B 0,C 180,E1 -9562.965,E2 -9562.965} C_VEL
LIN {X 0,Y 432.355,Z 468.251,A -85,B 0,C 180,E1 -9566.033,E2 -9566.033} C_VEL
LIN {X 0,Y 432.343,Z 468.251,A -85,B 0,C 180,E1 -9569.188,E2 -9569.188} C_VEL
LIN {X 0,Y 432.324,Z 468.259,A -85,B 0,C 180,E1 -9572.296,E2 -9572.296} C_VEL
LIN {X 0,Y 432.333,Z 468.258,A -85,B 0,C 180,E1 -9574.678,E2 -9574.678} C_VEL
LIN {X 0,Y 432.346,Z 468.253,A -85,B 0,C 180,E1 -9578.149,E2 -9578.149} C_VEL
LIN {X 0,Y 432.359,Z 468.252,A -85,B 0,C 180,E1 -9581.608,E2 -9581.608} C_VEL
LIN {X 0,Y 432.372,Z 468.249,A -85,B 0,C 180,E1 -9585.66,E2 -9585.66} C_VEL
LIN {X 0,Y 432.367,Z 468.253,A -85,B 0,C 180,E1 -9588.393,E2 -9588.393} C_VEL
LIN {X 0,Y 432.349,Z 468.254,A -85,B 0,C 180,E1 -9591.853,E2 -9591.853} C_VEL
LIN {X 0,Y 432.337,Z 468.254,A -85,B 0,C 180,E1 -9595.325,E2 -9595.325} C_VEL
LIN {X 0,Y 432.327,Z 468.255,A -85,B 0,C 180,E1 -9598.656,E2 -9598.656} C_VEL
LIN {X 0,Y 432.425,Z 468.441,A -85,B 0,C 180,E1 -9601.752,E2 -9601.752} C_VEL
LIN {X 0,Y 434.918,Z 479.34,A -85,B 0,C 180,E1 -9604.133,E2 -9604.133} C_VEL
LIN {X 0,Y 436.363,Z 487.035,A -85,B 0,C 180,E1 -9605.753,E2 -9605.753} C_VEL
LIN {X 0,Y 435.454,Z 501.226,A -85,B 0,C 180,E1 -9608.46,E2 -9608.46} C_VEL
LIN {X 0,Y 434.553,Z 516.13,A -85,B 0,C 180,E1 -9611.217,E2 -9611.217} C_VEL
LIN {X 0,Y 438.451,Z 536.187,A -85,B 0,C 180,E1 -9611.727,E2 -9611.727} C_VEL
LIN {X 0,Y 437.741,Z 628.234,A -85,B 0,C 180,E1 -9613.144,E2 -9613.144} C_VEL
LIN {X 0,Y 437.382,Z 641.803,A -85,B 0,C 180,E1 -9613.55,E2 -9613.55} C_VEL
LIN {X 0,Y 436.843,Z 654.583,A -85,B 0,C 180,E1 -9614.129,E2 -9614.129} C_VEL
LIN {X 0,Y 436.357,Z 664.758,A -85,B 0,C 180,E1 -9614.754,E2 -9614.754} C_VEL
LIN {X 0,Y 435.378,Z 669.978,A -85,B 0,C 180,E1 -9615.099,E2 -9615.099} C_VEL
LIN {X 0,Y 432.007,Z 678.249,A -85,B 0,C 180,E1 -9615.677,E2 -9615.677} C_VEL
LIN {X 0,Y 428.632,Z 686.056,A -85,B 0,C 180,E1 -9616.353,E2 -9616.353} C_VEL
LIN {X 0,Y 427.653,Z 690.543,A -85,B 0,C 180,E1 -9616.848,E2 -9616.848} C_VEL
LIN {X 0,Y 426.923,Z 700.026,A -85,B 0,C 180,E1 -9618.127,E2 -9618.127} C_VEL
LIN {X 0,Y 426.186,Z 708.557,A -85,B 0,C 180,E1 -9619.55,E2 -9619.55} C_VEL
LIN {X 0,Y 425.511,Z 715.424,A -85,B 0,C 180,E1 -9620.974,E2 -9620.974} C_VEL
LIN {X 0,Y 425.015,Z 720.92,A -85,B 0,C 180,E1 -9622.4,E2 -9622.4} C_VEL
LIN {X 0,Y 424.723,Z 725.264,A -85,B 0,C 180,E1 -9623.827,E2 -9623.827} C_VEL
LIN {X 0,Y 424.506,Z 728.582,A -85,B 0,C 180,E1 -9625.253,E2 -9625.253} C_VEL
LIN {X 0,Y 424.488,Z 730.273,A -85,B 0,C 180,E1 -9626.204,E2 -9626.204} C_VEL
LIN {X 0,Y 424.274,Z 732.487,A -85,B 0,C 180,E1 -9628.103,E2 -9628.103} C_VEL
LIN {X 0,Y 424.206,Z 733.267,A -85,B 0,C 180,E1 -9630.001,E2 -9630.001} C_VEL
LIN {X 0,Y 424.274,Z 732.557,A -85,B 0,C 180,E1 -9631.9,E2 -9631.9} C_VEL
LIN {X 0,Y 424.478,Z 730.401,A -85,B 0,C 180,E1 -9633.799,E2 -9633.799} C_VEL
LIN {X 0,Y 424.474,Z 727.766,A -85,B 0,C 180,E1 -9635.226,E2 -9635.226} C_VEL
LIN {X 0,Y 424.877,Z 724.166,A -85,B 0,C 180,E1 -9636.65,E2 -9636.65} C_VEL
LIN {X 0,Y 425.17,Z 719.528,A -85,B 0,C 180,E1 -9638.078,E2 -9638.078} C_VEL
LIN {X 0,Y 425.719,Z 713.686,A -85,B 0,C 180,E1 -9639.503,E2 -9639.503} C_VEL
LIN {X 0,Y 426.333,Z 706.439,A -85,B 0,C 180,E1 -9640.929,E2 -9640.929} C_VEL
LIN {X 0,Y 426.95,Z 699.05,A -85,B 0,C 180,E1 -9642.116,E2 -9642.116} C_VEL
LIN {X 0,Y 427.733,Z 690.11,A -85,B 0,C 180,E1 -9643.3,E2 -9643.3} C_VEL
LIN {X 0,Y 428.578,Z 680.081,A -85,B 0,C 180,E1 -9644.373,E2 -9644.373} C_VEL
LIN {X 0,Y 429.24,Z 669.211,A -85,B 0,C 180,E1 -9645.31,E2 -9645.31} C_VEL
LIN {X 0,Y 430.019,Z 656.839,A -85,B 0,C 180,E1 -9646.132,E2 -9646.132} C_VEL
LIN {X 0,Y 430.556,Z 644.971,A -85,B 0,C 180,E1 -9646.721,E2 -9646.721} C_VEL
LIN {X 0,Y 430.984,Z 631.832,A -85,B 0,C 180,E1 -9647.162,E2 -9647.162} C_VEL
LIN {X 0,Y 431.223,Z 614.07,A -85,B 0,C 180,E1 -9647.488,E2 -9647.488} C_VEL
LIN {X 0,Y 431.819,Z 537.188,A -85,B 0,C 180,E1 -9648.669,E2 -9648.669} C_VEL
LIN {X 0,Y 427.732,Z 516.001,A -85,B 0,C 180,E1 -9649.248,E2 -9649.248} C_VEL
LIN {X 0,Y 428.893,Z 498.003,A -85,B 0,C 180,E1 -9652.65,E2 -9652.65} C_VEL
LIN {X 0,Y 429.551,Z 488.973,A -85,B 0,C 180,E1 -9654.402,E2 -9654.402} C_VEL
LIN {X 0,Y 427.352,Z 477.743,A -85,B 0,C 180,E1 -9656.816,E2 -9656.816} C_VEL
LIN {X 0,Y 425.348,Z 469.135,A -85,B 0,C 180,E1 -9658.772,E2 -9658.772} C_VEL
LIN {X 0,Y 425.271,Z 469.142,A -85,B 0,C 180,E1 -9661.927,E2 -9661.927} C_VEL
LIN {X 0,Y 425.305,Z 469.133,A -85,B 0,C 180,E1 -9665.336,E2 -9665.336} C_VEL
LIN {X 0,Y 425.31,Z 469.128,A -85,B 0,C 180,E1 -9669.045,E2 -9669.045} C_VEL
LIN {X 0,Y 425.285,Z 469.134,A -85,B 0,C 180,E1 -9672.653,E2 -9672.653} C_VEL
LIN {X 0,Y 425.268,Z 469.137,A -85,B 0,C 180,E1 -9676.045,E2 -9676.045} C_VEL
LIN {X 0,Y 425.28,Z 469.13,A -85,B 0,C 180,E1 -9678.622,E2 -9678.622} C_VEL
LIN {X 0,Y 425.306,Z 469.129,A -85,B 0,C 180,E1 -9681.102,E2 -9681.102} C_VEL
LIN {X 0,Y 425.307,Z 469.129,A -85,B 0,C 180,E1 -9684.665,E2 -9684.665} C_VEL
LIN {X 0,Y 425.271,Z 469.138,A -85,B 0,C 180,E1 -9688.073,E2 -9688.073} C_VEL
LIN {X 0,Y 425.392,Z 469.262,A -85,B 0,C 180,E1 -9691.742,E2 -9691.742} C_VEL
LIN {X 0,Y 428.869,Z 485.297,A -85,B 0,C 180,E1 -9694.572,E2 -9694.572} C_VEL
LIN {X 0,Y 429.15,Z 489.735,A -85,B 0,C 180,E1 -9695.317,E2 -9695.317} C_VEL
LIN {X 0,Y 428.262,Z 510.004,A -85,B 0,C 180,E1 -9698.584,E2 -9698.584} C_VEL
LIN {X 0,Y 427.575,Z 528.65,A -85,B 0,C 180,E1 -9701.579,E2 -9701.579} C_VEL
LIN {X 0,Y 430.266,Z 545.796,A -85,B 0,C 180,E1 -9702.033,E2 -9702.033} C_VEL
LIN {X 0,Y 428.716,Z 637.953,A -85,B 0,C 180,E1 -9703.849,E2 -9703.849} C_VEL
LIN {X 0,Y 428.435,Z 651.616,A -85,B 0,C 180,E1 -9704.296,E2 -9704.296} C_VEL
LIN {X 0,Y 427.897,Z 664.959,A -85,B 0,C 180,E1 -9704.947,E2 -9704.947} C_VEL
LIN {X 0,Y 427.412,Z 676.834,A -85,B 0,C 180,E1 -9705.721,E2 -9705.721} C_VEL
LIN {X 0,Y 426.888,Z 688.19,A -85,B 0,C 180,E1 -9706.674,E2 -9706.674} C_VEL
LIN {X 0,Y 426.287,Z 698.483,A -85,B 0,C 180,E1 -9707.745,E2 -9707.745} C_VEL
LIN {X 0,Y 425.809,Z 706.959,A -85,B 0,C 180,E1 -9708.817,E2 -9708.817} C_VEL
LIN {X 0,Y 425.41,Z 714.783,A -85,B 0,C 180,E1 -9710.01,E2 -9710.01} C_VEL
LIN {X 0,Y 424.965,Z 722.392,A -85,B 0,C 180,E1 -9711.44,E2 -9711.44} C_VEL
LIN {X 0,Y 424.62,Z 728.683,A -85,B 0,C 180,E1 -9712.917,E2 -9712.917} C_VEL
LIN {X 0,Y 424.488,Z 733.314,A -85,B 0,C 180,E1 -9714.299,E2 -9714.299} C_VEL
LIN {X 0,Y 424.303,Z 736.976,A -85,B 0,C 180,E1 -9715.725,E2 -9715.725} C_VEL
LIN {X 0,Y 424.293,Z 739.581,A -85,B 0,C 180,E1 -9717.152,E2 -9717.152} C_VEL
LIN {X 0,Y 424.196,Z 740.774,A -85,B 0,C 180,E1 -9718.101,E2 -9718.101} C_VEL
LIN {X 0,Y 424.141,Z 741.52,A -85,B 0,C 180,E1 -9719.05,E2 -9719.05} C_VEL
LIN {X 0,Y 424.135,Z 741.869,A -85,B 0,C 180,E1 -9720,E2 -9720} C_VEL
LIN {X 0,Y 424.167,Z 741.799,A -85,B 0,C 180,E1 -9720.949,E2 -9720.949} C_VEL
LIN {X 0,Y 424.217,Z 741.268,A -85,B 0,C 180,E1 -9721.899,E2 -9721.899} C_VEL
LIN {X 0,Y 424.305,Z 740.333,A -85,B 0,C 180,E1 -9722.848,E2 -9722.848} C_VEL
LIN {X 0,Y 424.421,Z 738.985,A -85,B 0,C 180,E1 -9723.798,E2 -9723.798} C_VEL
LIN {X 0,Y 424.405,Z 736.102,A -85,B 0,C 180,E1 -9725.226,E2 -9725.226} C_VEL
LIN {X 0,Y 424.726,Z 732.116,A -85,B 0,C 180,E1 -9726.651,E2 -9726.651} C_VEL
LIN {X 0,Y 424.955,Z 726.932,A -85,B 0,C 180,E1 -9728.081,E2 -9728.081} C_VEL
LIN {X 0,Y 425.438,Z 720.395,A -85,B 0,C 180,E1 -9729.508,E2 -9729.508} C_VEL
LIN {X 0,Y 425.936,Z 712.268,A -85,B 0,C 180,E1 -9730.938,E2 -9730.938} C_VEL
LIN {X 0,Y 426.478,Z 703.874,A -85,B 0,C 180,E1 -9732.129,E2 -9732.129} C_VEL
LIN {X 0,Y 427.156,Z 693.554,A -85,B 0,C 180,E1 -9733.317,E2 -9733.317} C_VEL
LIN {X 0,Y 427.735,Z 683.387,A -85,B 0,C 180,E1 -9734.268,E2 -9734.268} C_VEL
LIN {X 0,Y 428.276,Z 672.23,A -85,B 0,C 180,E1 -9735.1,E2 -9735.1} C_VEL
LIN {X 0,Y 428.837,Z 659.877,A -85,B 0,C 180,E1 -9735.811,E2 -9735.811} C_VEL
LIN {X 0,Y 429.307,Z 647.282,A -85,B 0,C 180,E1 -9736.342,E2 -9736.342} C_VEL
LIN {X 0,Y 429.667,Z 633.087,A -85,B 0,C 180,E1 -9736.725,E2 -9736.725} C_VEL
LIN {X 0,Y 431.559,Z 549.34,A -85,B 0,C 180,E1 -9738.509,E2 -9738.509} C_VEL
LIN {X 0,Y 431.42,Z 544.768,A -85,B 0,C 180,E1 -9738.626,E2 -9738.626} C_VEL
LIN {X 0,Y 428.809,Z 531.025,A -85,B 0,C 180,E1 -9739.135,E2 -9739.135} C_VEL
LIN {X 0,Y 429.672,Z 510.744,A -85,B 0,C 180,E1 -9742.352,E2 -9742.352} C_VEL
LIN {X 0,Y 430.577,Z 492.12,A -85,B 0,C 180,E1 -9745.299,E2 -9745.299} C_VEL
LIN {X 0,Y 429.996,Z 486.791,A -85,B 0,C 180,E1 -9746.187,E2 -9746.187} C_VEL
LIN {X 0,Y 427.34,Z 475.666,A -85,B 0,C 180,E1 -9748.217,E2 -9748.217} C_VEL
LIN {X 0,Y 425.291,Z 469.139,A -85,B 0,C 180,E1 -9749.487,E2 -9749.487} C_VEL
LIN {X 0,Y 425.287,Z 469.136,A -85,B 0,C 180,E1 -9753.047,E2 -9753.047} C_VEL
LIN {X 0,Y 425.29,Z 469.135,A -85,B 0,C 180,E1 -9755.929,E2 -9755.929} C_VEL
LIN {X 0,Y 425.308,Z 469.13,A -85,B 0,C 180,E1 -9759.044,E2 -9759.044} C_VEL
LIN {X 0,Y 425.279,Z 469.136,A -85,B 0,C 180,E1 -9762.652,E2 -9762.652} C_VEL
LIN {X 0,Y 425.266,Z 469.14,A -85,B 0,C 180,E1 -9766.044,E2 -9766.044} C_VEL
LIN {X 0,Y 425.278,Z 469.133,A -85,B 0,C 180,E1 -9768.621,E2 -9768.621} C_VEL
LIN {X 0,Y 425.301,Z 469.13,A -85,B 0,C 180,E1 -9771.101,E2 -9771.101} C_VEL
LIN {X 0,Y 425.304,Z 469.132,A -85,B 0,C 180,E1 -9774.663,E2 -9774.663} C_VEL
LIN {X 0,Y 425.27,Z 469.139,A -85,B 0,C 180,E1 -9778.072,E2 -9778.072} C_VEL
LIN {X 0,Y 425.324,Z 469.325,A -85,B 0,C 180,E1 -9779.082,E2 -9779.082} C_VEL
LIN {X 0,Y 429.305,Z 484.558,A -85,B 0,C 180,E1 -9781.845,E2 -9781.845} C_VEL
LIN {X 0,Y 431.251,Z 493.184,A -85,B 0,C 180,E1 -9783.335,E2 -9783.335} C_VEL
LIN {X 0,Y 431.209,Z 496.773,A -85,B 0,C 180,E1 -9783.891,E2 -9783.891} C_VEL
LIN {X 0,Y 429.668,Z 515.236,A -85,B 0,C 180,E1 -9786.664,E2 -9786.664} C_VEL
LIN {X 0,Y 429.133,Z 522.929,A -85,B 0,C 180,E1 -9787.788,E2 -9787.788} C_VEL
LIN {X 0,Y 432.567,Z 546.423,A -85,B 0,C 180,E1 -9788.387,E2 -9788.387} C_VEL
LIN {X 0,Y 430.776,Z 657.857,A -85,B 0,C 180,E1 -9790.398,E2 -9790.398} C_VEL
LIN {X 0,Y 430.256,Z 672.102,A -85,B 0,C 180,E1 -9790.838,E2 -9790.838} C_VEL
LIN {X 0,Y 429.55,Z 685.71,A -85,B 0,C 180,E1 -9791.443,E2 -9791.443} C_VEL
LIN {X 0,Y 428.803,Z 698.903,A -85,B 0,C 180,E1 -9792.225,E2 -9792.225} C_VEL
LIN {X 0,Y 428.03,Z 711.542,A -85,B 0,C 180,E1 -9793.177,E2 -9793.177} C_VEL
LIN {X 0,Y 427.13,Z 723.093,A -85,B 0,C 180,E1 -9794.246,E2 -9794.246} C_VEL
LIN {X 0,Y 426.384,Z 733.72,A -85,B 0,C 180,E1 -9795.441,E2 -9795.441} C_VEL
LIN {X 0,Y 425.764,Z 742.628,A -85,B 0,C 180,E1 -9796.637,E2 -9796.637} C_VEL
LIN {X 0,Y 425.233,Z 751.626,A -85,B 0,C 180,E1 -9798.076,E2 -9798.076} C_VEL
LIN {X 0,Y 424.728,Z 760.238,A -85,B 0,C 180,E1 -9799.752,E2 -9799.752} C_VEL
LIN {X 0,Y 424.425,Z 767.13,A -85,B 0,C 180,E1 -9801.428,E2 -9801.428} C_VEL
LIN {X 0,Y 424.295,Z 773.232,A -85,B 0,C 180,E1 -9803.341,E2 -9803.341} C_VEL
LIN {X 0,Y 424.215,Z 777.673,A -85,B 0,C 180,E1 -9805.247,E2 -9805.247} C_VEL
LIN {X 0,Y 424.259,Z 780.59,A -85,B 0,C 180,E1 -9807.15,E2 -9807.15} C_VEL
LIN {X 0,Y 424.188,Z 782.041,A -85,B 0,C 180,E1 -9809.049,E2 -9809.049} C_VEL
LIN {X 0,Y 424.187,Z 782.042,A -85,B 0,C 180,E1 -9810.948,E2 -9810.948} C_VEL
LIN {X 0,Y 424.258,Z 780.593,A -85,B 0,C 180,E1 -9812.847,E2 -9812.847} C_VEL
LIN {X 0,Y 424.214,Z 777.678,A -85,B 0,C 180,E1 -9814.75,E2 -9814.75} C_VEL
LIN {X 0,Y 424.293,Z 773.231,A -85,B 0,C 180,E1 -9816.657,E2 -9816.657} C_VEL
LIN {X 0,Y 424.422,Z 767.127,A -85,B 0,C 180,E1 -9818.569,E2 -9818.569} C_VEL
LIN {X 0,Y 424.727,Z 760.237,A -85,B 0,C 180,E1 -9820.245,E2 -9820.245} C_VEL
LIN {X 0,Y 425.229,Z 751.623,A -85,B 0,C 180,E1 -9821.921,E2 -9821.921} C_VEL
LIN {X 0,Y 425.764,Z 742.623,A -85,B 0,C 180,E1 -9823.36,E2 -9823.36} C_VEL
LIN {X 0,Y 426.503,Z 731.715,A -85,B 0,C 180,E1 -9824.797,E2 -9824.797} C_VEL
LIN {X 0,Y 427.26,Z 720.688,A -85,B 0,C 180,E1 -9825.992,E2 -9825.992} C_VEL
LIN {X 0,Y 428.154,Z 708.637,A -85,B 0,C 180,E1 -9827.061,E2 -9827.061} C_VEL
LIN {X 0,Y 428.998,Z 695.286,A -85,B 0,C 180,E1 -9828.011,E2 -9828.011} C_VEL
LIN {X 0,Y 429.742,Z 681.765,A -85,B 0,C 180,E1 -9828.75,E2 -9828.75} C_VEL
LIN {X 0,Y 430.441,Z 666.993,A -85,B 0,C 180,E1 -9829.337,E2 -9829.337} C_VEL
LIN {X 0,Y 430.963,Z 652.238,A -85,B 0,C 180,E1 -9829.715,E2 -9829.715} C_VEL
LIN {X 0,Y 432.506,Z 545.64,A -85,B 0,C 180,E1 -9831.624,E2 -9831.624} C_VEL
LIN {X 0,Y 429.085,Z 522.515,A -85,B 0,C 180,E1 -9832.224,E2 -9832.224} C_VEL
LIN {X 0,Y 430.942,Z 500.074,A -85,B 0,C 180,E1 -9835.604,E2 -9835.604} C_VEL
LIN {X 0,Y 431.24,Z 493.222,A -85,B 0,C 180,E1 -9836.652,E2 -9836.652} C_VEL
LIN {X 0,Y 427.882,Z 478.936,A -85,B 0,C 180,E1 -9839.147,E2 -9839.147} C_VEL
LIN {X 0,Y 425.28,Z 469.135,A -85,B 0,C 180,E1 -9840.953,E2 -9840.953} C_VEL
LIN {X 0,Y 425.306,Z 469.118,A -85,B 0,C 180,E1 -9844.287,E2 -9844.287} C_VEL
LIN {X 0,Y 425.283,Z 469.134,A -85,B 0,C 180,E1 -9847.692,E2 -9847.692} C_VEL
LIN {X 0,Y 425.296,Z 469.135,A -85,B 0,C 180,E1 -9850.523,E2 -9850.523} C_VEL
LIN {X 0,Y 425.309,Z 469.13,A -85,B 0,C 180,E1 -9853.358,E2 -9853.358} C_VEL
LIN {X 0,Y 425.324,Z 469.131,A -85,B 0,C 180,E1 -9856.637,E2 -9856.637} C_VEL
LIN {X 0,Y 425.303,Z 469.127,A -85,B 0,C 180,E1 -9859.875,E2 -9859.875} C_VEL
LIN {X 0,Y 425.278,Z 469.13,A -85,B 0,C 180,E1 -9862.486,E2 -9862.486} C_VEL
LIN {X 0,Y 425.298,Z 469.124,A -85,B 0,C 180,E1 -9865.817,E2 -9865.817} C_VEL
LIN {X 0,Y 425.294,Z 469.13,A -85,B 0,C 180,E1 -9869.235,E2 -9869.235} C_VEL
LIN {X 0,Y 425.34,Z 469.125,A -85,B 0,C 180,E1 -9872.442,E2 -9872.442} C_VEL
LIN {X 0,Y 425.34,Z 469.121,A -85,B 0,C 180,E1 -9875.602,E2 -9875.602} C_VEL
LIN {X 0,Y 425.282,Z 469.116,A -85,B 0,C 180,E1 -9878.681,E2 -9878.681} C_VEL
LIN {X 0,Y 425.322,Z 469.127,A -85,B 0,C 180,E1 -9881.702,E2 -9881.702} C_VEL
LIN {X 0,Y 425.338,Z 469.125,A -85,B 0,C 180,E1 -9884.67,E2 -9884.67} C_VEL
LIN {X 0,Y 425.421,Z 469.113,A -85,B 0,C 180,E1 -9887.599,E2 -9887.599} C_VEL
LIN {X 0,Y 425.431,Z 469.113,A -85,B 0,C 180,E1 -9891.45,E2 -9891.45} C_VEL
LIN {X 0,Y 425.546,Z 469.095,A -85,B 0,C 180,E1 -9894.313,E2 -9894.313} C_VEL
LIN {X 0,Y 425.565,Z 469.096,A -85,B 0,C 180,E1 -9898.107,E2 -9898.107} C_VEL
LIN {X 0,Y 425.693,Z 469.079,A -85,B 0,C 180,E1 -9900,E2 -9900} C_VEL
LIN {X 0,Y 425.547,Z 469.095,A -85,B 0,C 180,E1 -9902.84,E2 -9902.84} C_VEL
LIN {X 0,Y 425.519,Z 469.106,A -85,B 0,C 180,E1 -9906.649,E2 -9906.649} C_VEL
LIN {X 0,Y 425.393,Z 469.116,A -85,B 0,C 180,E1 -9909.51,E2 -9909.51} C_VEL
LIN {X 0,Y 425.393,Z 469.115,A -85,B 0,C 180,E1 -9912.911,E2 -9912.911} C_VEL
LIN {X 0,Y 425.359,Z 469.124,A -85,B 0,C 180,E1 -9916.61,E2 -9916.61} C_VEL
LIN {X 0,Y 425.318,Z 469.127,A -85,B 0,C 180,E1 -9919.637,E2 -9919.637} C_VEL
LIN {X 0,Y 425.297,Z 469.129,A -85,B 0,C 180,E1 -9923.366,E2 -9923.366} C_VEL
LIN {X 0,Y 425.339,Z 469.126,A -85,B 0,C 180,E1 -9926.846,E2 -9926.846} C_VEL
LIN {X 0,Y 425.309,Z 469.127,A -85,B 0,C 180,E1 -9929.718,E2 -9929.718} C_VEL
LIN {X 0,Y 425.276,Z 469.131,A -85,B 0,C 180,E1 -9933.049,E2 -9933.049} C_VEL
LIN {X 0,Y 425.277,Z 469.135,A -85,B 0,C 180,E1 -9935.93,E2 -9935.93} C_VEL
LIN {X 0,Y 425.306,Z 469.131,A -85,B 0,C 180,E1 -9939.047,E2 -9939.047} C_VEL
LIN {X 0,Y 425.308,Z 469.132,A -85,B 0,C 180,E1 -9941.963,E2 -9941.963} C_VEL
LIN {X 0,Y 425.306,Z 469.129,A -85,B 0,C 180,E1 -9945.281,E2 -9945.281} C_VEL
LIN {X 0,Y 425.305,Z 469.134,A -85,B 0,C 180,E1 -9948.627,E2 -9948.627} C_VEL
LIN {X 0,Y 425.32,Z 469.13,A -85,B 0,C 180,E1 -9951.106,E2 -9951.106} C_VEL
LIN {X 0,Y 425.297,Z 469.136,A -85,B 0,C 180,E1 -9954.666,E2 -9954.666} C_VEL
LIN {X 0,Y 425.27,Z 469.137,A -85,B 0,C 180,E1 -9958.075,E2 -9958.075} C_VEL
LIN {X 0,Y 425.352,Z 469.196,A -85,B 0,C 180,E1 -9961.371,E2 -9961.371} C_VEL
LIN {X 0,Y 427.967,Z 480.605,A -85,B 0,C 180,E1 -9963.909,E2 -9963.909} C_VEL
LIN {X 0,Y 429.472,Z 488.479,A -85,B 0,C 180,E1 -9965.596,E2 -9965.596} C_VEL
LIN {X 0,Y 428.667,Z 501.406,A -85,B 0,C 180,E1 -9968.102,E2 -9968.102} C_VEL
LIN {X 0,Y 427.706,Z 516.141,A -85,B 0,C 180,E1 -9970.874,E2 -9970.874} C_VEL
LIN {X 0,Y 431.804,Z 537.897,A -85,B 0,C 180,E1 -9971.435,E2 -9971.435} C_VEL
LIN {X 0,Y 431.024,Z 628.243,A -85,B 0,C 180,E1 -9972.842,E2 -9972.842} C_VEL
LIN {X 0,Y 430.727,Z 641.126,A -85,B 0,C 180,E1 -9973.227,E2 -9973.227} C_VEL
LIN {X 0,Y 430.094,Z 654.177,A -85,B 0,C 180,E1 -9973.812,E2 -9973.812} C_VEL
LIN {X 0,Y 429.467,Z 666.457,A -85,B 0,C 180,E1 -9974.58,E2 -9974.58} C_VEL
LIN {X 0,Y 428.781,Z 676.969,A -85,B 0,C 180,E1 -9975.431,E2 -9975.431} C_VEL
LIN {X 0,Y 427.856,Z 688.303,A -85,B 0,C 180,E1 -9976.585,E2 -9976.585} C_VEL
LIN {X 0,Y 427.653,Z 690.543,A -85,B 0,C 180,E1 -9976.848,E2 -9976.848} C_VEL
LIN {X 0,Y 426.688,Z 694.901,A -85,B 0,C 180,E1 -9977.374,E2 -9977.374} C_VEL
LIN {X 0,Y 421.864,Z 704.215,A -85,B 0,C 180,E1 -9978.603,E2 -9978.603} C_VEL
LIN {X 0,Y 419.525,Z 709.053,A -85,B 0,C 180,E1 -9979.394,E2 -9979.394} C_VEL
LIN {X 0,Y 419.008,Z 711.29,A -85,B 0,C 180,E1 -9979.827,E2 -9979.827} C_VEL
LIN {X 0,Y 418.323,Z 717.806,A -85,B 0,C 180,E1 -9981.305,E2 -9981.305} C_VEL
LIN {X 0,Y 417.84,Z 723.42,A -85,B 0,C 180,E1 -9982.92,E2 -9982.92} C_VEL
LIN {X 0,Y 417.528,Z 726.88,A -85,B 0,C 180,E1 -9984.205,E2 -9984.205} C_VEL
LIN {X 0,Y 417.427,Z 729,A -85,B 0,C 180,E1 -9985.172,E2 -9985.172} C_VEL
LIN {X 0,Y 417.431,Z 730.685,A -85,B 0,C 180,E1 -9986.14,E2 -9986.14} C_VEL
LIN {X 0,Y 417.197,Z 732.897,A -85,B 0,C 180,E1 -9988.071,E2 -9988.071} C_VEL
LIN {X 0,Y 417.12,Z 733.676,A -85,B 0,C 180,E1 -9990.001,E2 -9990.001} C_VEL
LIN {X 0,Y 417.197,Z 732.967,A -85,B 0,C 180,E1 -9991.932,E2 -9991.932} C_VEL
LIN {X 0,Y 417.422,Z 730.812,A -85,B 0,C 180,E1 -9993.863,E2 -9993.863} C_VEL
LIN {X 0,Y 417.417,Z 728.182,A -85,B 0,C 180,E1 -9995.315,E2 -9995.315} C_VEL
LIN {X 0,Y 417.818,Z 724.589,A -85,B 0,C 180,E1 -9996.763,E2 -9996.763} C_VEL
LIN {X 0,Y 418.145,Z 719.957,A -85,B 0,C 180,E1 -9998.215,E2 -9998.215} C_VEL
LIN {X 0,Y 418.833,Z 713.049,A -85,B 0,C 180,E1 -9999.905,E2 -9999.905} C_VEL
LIN {X 0,Y 419.519,Z 705.532,A -85,B 0,C 180,E1 -10001.354,E2 -10001.354} C_VEL
LIN {X 0,Y 420.357,Z 696.145,A -85,B 0,C 180,E1 -10002.8,E2 -10002.8} C_VEL
LIN {X 0,Y 421.249,Z 686.454,A -85,B 0,C 180,E1 -10004.001,E2 -10004.001} C_VEL
LIN {X 0,Y 421.951,Z 676.829,A -85,B 0,C 180,E1 -10004.972,E2 -10004.972} C_VEL
LIN {X 0,Y 422.676,Z 666.653,A -85,B 0,C 180,E1 -10005.801,E2 -10005.801} C_VEL
LIN {X 0,Y 423.459,Z 654.317,A -85,B 0,C 180,E1 -10006.575,E2 -10006.575} C_VEL
LIN {X 0,Y 423.971,Z 641.996,A -85,B 0,C 180,E1 -10007.144,E2 -10007.144} C_VEL
LIN {X 0,Y 424.368,Z 629.397,A -85,B 0,C 180,E1 -10007.531,E2 -10007.531} C_VEL
LIN {X 0,Y 424.79,Z 586.329,A -85,B 0,C 180,E1 -10008.229,E2 -10008.229} C_VEL
LIN {X 0,Y 425.02,Z 537.531,A -85,B 0,C 180,E1 -10009.002,E2 -10009.002} C_VEL
LIN {X 0,Y 420.892,Z 516.198,A -85,B 0,C 180,E1 -10009.574,E2 -10009.574} C_VEL
LIN {X 0,Y 422.108,Z 498.178,A -85,B 0,C 180,E1 -10013.035,E2 -10013.035} C_VEL
LIN {X 0,Y 422.687,Z 490.41,A -85,B 0,C 180,E1 -10014.563,E2 -10014.563} C_VEL
LIN {X 0,Y 419.965,Z 477.007,A -85,B 0,C 180,E1 -10017.508,E2 -10017.508} C_VEL
LIN {X 0,Y 418.271,Z 470.019,A -85,B 0,C 180,E1 -10019.163,E2 -10019.163} C_VEL
LIN {X 0,Y 418.264,Z 470.01,A -85,B 0,C 180,E1 -10022.845,E2 -10022.845} C_VEL
LIN {X 0,Y 418.254,Z 470.009,A -85,B 0,C 180,E1 -10026.239,E2 -10026.239} C_VEL
LIN {X 0,Y 418.262,Z 470.013,A -85,B 0,C 180,E1 -10029.682,E2 -10029.682} C_VEL
LIN {X 0,Y 418.239,Z 470.012,A -85,B 0,C 180,E1 -10032.322,E2 -10032.322} C_VEL
LIN {X 0,Y 418.244,Z 470.007,A -85,B 0,C 180,E1 -10035.109,E2 -10035.109} C_VEL
LIN {X 0,Y 418.246,Z 470.007,A -85,B 0,C 180,E1 -10037.767,E2 -10037.767} C_VEL
LIN {X 0,Y 418.258,Z 470.005,A -85,B 0,C 180,E1 -10041.558,E2 -10041.558} C_VEL
LIN {X 0,Y 418.266,Z 470.008,A -85,B 0,C 180,E1 -10045.159,E2 -10045.159} C_VEL
LIN {X 0,Y 418.252,Z 470.013,A -85,B 0,C 180,E1 -10047.472,E2 -10047.472} C_VEL
LIN {X 0,Y 418.275,Z 470.008,A -85,B 0,C 180,E1 -10050.896,E2 -10050.896} C_VEL
LIN {X 0,Y 418.343,Z 470.192,A -85,B 0,C 180,E1 -10051.496,E2 -10051.496} C_VEL
LIN {X 0,Y 421.637,Z 485.184,A -85,B 0,C 180,E1 -10054.172,E2 -10054.172} C_VEL
LIN {X 0,Y 422.269,Z 489.313,A -85,B 0,C 180,E1 -10054.887,E2 -10054.887} C_VEL
LIN {X 0,Y 421.41,Z 509.752,A -85,B 0,C 180,E1 -10058.218,E2 -10058.218} C_VEL
LIN {X 0,Y 420.651,Z 529.005,A -85,B 0,C 180,E1 -10061.318,E2 -10061.318} C_VEL
LIN {X 0,Y 423.414,Z 547.308,A -85,B 0,C 180,E1 -10061.815,E2 -10061.815} C_VEL
LIN {X 0,Y 421.757,Z 638.99,A -85,B 0,C 180,E1 -10063.668,E2 -10063.668} C_VEL
LIN {X 0,Y 421.507,Z 651.612,A -85,B 0,C 180,E1 -10064.093,E2 -10064.093} C_VEL
LIN {X 0,Y 420.961,Z 665.033,A -85,B 0,C 180,E1 -10064.755,E2 -10064.755} C_VEL
LIN {X 0,Y 420.433,Z 677.319,A -85,B 0,C 180,E1 -10065.568,E2 -10065.568} C_VEL
LIN {X 0,Y 419.863,Z 688.989,A -85,B 0,C 180,E1 -10066.57,E2 -10066.57} C_VEL
LIN {X 0,Y 419.247,Z 699.216,A -85,B 0,C 180,E1 -10067.659,E2 -10067.659} C_VEL
LIN {X 0,Y 418.739,Z 708.462,A -85,B 0,C 180,E1 -10068.871,E2 -10068.871} C_VEL
LIN {X 0,Y 418.212,Z 717.436,A -85,B 0,C 180,E1 -10070.325,E2 -10070.325} C_VEL
LIN {X 0,Y 417.811,Z 724.642,A -85,B 0,C 180,E1 -10071.78,E2 -10071.78} C_VEL
LIN {X 0,Y 417.526,Z 730.503,A -85,B 0,C 180,E1 -10073.279,E2 -10073.279} C_VEL
LIN {X 0,Y 417.339,Z 734.817,A -85,B 0,C 180,E1 -10074.685,E2 -10074.685} C_VEL
LIN {X 0,Y 417.218,Z 738.168,A -85,B 0,C 180,E1 -10076.136,E2 -10076.136} C_VEL
LIN {X 0,Y 417.227,Z 739.834,A -85,B 0,C 180,E1 -10077.103,E2 -10077.103} C_VEL
LIN {X 0,Y 417.123,Z 741.068,A -85,B 0,C 180,E1 -10078.069,E2 -10078.069} C_VEL
LIN {X 0,Y 417.061,Z 741.837,A -85,B 0,C 180,E1 -10079.034,E2 -10079.034} C_VEL
LIN {X 0,Y 417.053,Z 742.205,A -85,B 0,C 180,E1 -10080,E2 -10080} C_VEL
LIN {X 0,Y 417.085,Z 742.161,A -85,B 0,C 180,E1 -10080.965,E2 -10080.965} C_VEL
LIN {X 0,Y 417.143,Z 741.65,A -85,B 0,C 180,E1 -10081.931,E2 -10081.931} C_VEL
LIN {X 0,Y 417.243,Z 740.728,A -85,B 0,C 180,E1 -10082.896,E2 -10082.896} C_VEL
LIN {X 0,Y 417.363,Z 739.4,A -85,B 0,C 180,E1 -10083.862,E2 -10083.862} C_VEL
LIN {X 0,Y 417.355,Z 736.555,A -85,B 0,C 180,E1 -10085.314,E2 -10085.314} C_VEL
LIN {X 0,Y 417.711,Z 732.063,A -85,B 0,C 180,E1 -10086.933,E2 -10086.933} C_VEL
LIN {X 0,Y 417.939,Z 727.472,A -85,B 0,C 180,E1 -10088.218,E2 -10088.218} C_VEL
LIN {X 0,Y 418.469,Z 720.954,A -85,B 0,C 180,E1 -10089.668,E2 -10089.668} C_VEL
LIN {X 0,Y 418.997,Z 712.846,A -85,B 0,C 180,E1 -10091.122,E2 -10091.122} C_VEL
LIN {X 0,Y 419.566,Z 704.489,A -85,B 0,C 180,E1 -10092.332,E2 -10092.332} C_VEL
LIN {X 0,Y 420.279,Z 694.218,A -85,B 0,C 180,E1 -10093.539,E2 -10093.539} C_VEL
LIN {X 0,Y 420.922,Z 684.164,A -85,B 0,C 180,E1 -10094.504,E2 -10094.504} C_VEL
LIN {X 0,Y 421.499,Z 673.216,A -85,B 0,C 180,E1 -10095.349,E2 -10095.349} C_VEL
LIN {X 0,Y 422.108,Z 661.114,A -85,B 0,C 180,E1 -10096.069,E2 -10096.069} C_VEL
LIN {X 0,Y 422.595,Z 648.127,A -85,B 0,C 180,E1 -10096.64,E2 -10096.64} C_VEL
LIN {X 0,Y 422.983,Z 634.297,A -85,B 0,C 180,E1 -10097.028,E2 -10097.028} C_VEL
LIN {X 0,Y 424.649,Z 563.675,A -85,B 0,C 180,E1 -10098.576,E2 -10098.576} C_VEL
LIN {X 0,Y 425.038,Z 546.207,A -85,B 0,C 180,E1 -10098.985,E2 -10098.985} C_VEL
LIN {X 0,Y 422.182,Z 531.521,A -85,B 0,C 180,E1 -10099.542,E2 -10099.542} C_VEL
LIN {X 0,Y 423.098,Z 511.745,A -85,B 0,C 180,E1 -10102.718,E2 -10102.718} C_VEL
LIN {X 0,Y 423.993,Z 494.171,A -85,B 0,C 180,E1 -10105.529,E2 -10105.529} C_VEL
LIN {X 0,Y 423.528,Z 489.424,A -85,B 0,C 180,E1 -10106.352,E2 -10106.352} C_VEL
LIN {X 0,Y 421.324,Z 479.873,A -85,B 0,C 180,E1 -10108.114,E2 -10108.114} C_VEL
LIN {X 0,Y 418.246,Z 470.017,A -85,B 0,C 180,E1 -10110.098,E2 -10110.098} C_VEL
LIN {X 0,Y 418.254,Z 470.012,A -85,B 0,C 180,E1 -10113.677,E2 -10113.677} C_VEL
LIN {X 0,Y 418.251,Z 470.01,A -85,B 0,C 180,E1 -10117.223,E2 -10117.223} C_VEL
LIN {X 0,Y 418.26,Z 470.012,A -85,B 0,C 180,E1 -10119.681,E2 -10119.681} C_VEL
LIN {X 0,Y 418.234,Z 470.014,A -85,B 0,C 180,E1 -10122.321,E2 -10122.321} C_VEL
LIN {X 0,Y 418.24,Z 470.012,A -85,B 0,C 180,E1 -10125.108,E2 -10125.108} C_VEL
LIN {X 0,Y 418.244,Z 470.013,A -85,B 0,C 180,E1 -10127.766,E2 -10127.766} C_VEL
LIN {X 0,Y 418.25,Z 470.007,A -85,B 0,C 180,E1 -10130.62,E2 -10130.62} C_VEL
LIN {X 0,Y 418.247,Z 470.011,A -85,B 0,C 180,E1 -10133.975,E2 -10133.975} C_VEL
LIN {X 0,Y 418.262,Z 470.011,A -85,B 0,C 180,E1 -10137.155,E2 -10137.155} C_VEL
LIN {X 0,Y 418.283,Z 470.15,A -85,B 0,C 180,E1 -10138.667,E2 -10138.667} C_VEL
LIN {X 0,Y 422.046,Z 484.478,A -85,B 0,C 180,E1 -10141.334,E2 -10141.334} C_VEL
LIN {X 0,Y 424.44,Z 494.911,A -85,B 0,C 180,E1 -10143.178,E2 -10143.178} C_VEL
LIN {X 0,Y 424.397,Z 498.244,A -85,B 0,C 180,E1 -10143.705,E2 -10143.705} C_VEL
LIN {X 0,Y 422.793,Z 516.433,A -85,B 0,C 180,E1 -10146.487,E2 -10146.487} C_VEL
LIN {X 0,Y 422.299,Z 522.54,A -85,B 0,C 180,E1 -10147.429,E2 -10147.429} C_VEL
LIN {X 0,Y 425.902,Z 546.857,A -85,B 0,C 180,E1 -10148.068,E2 -10148.068} C_VEL
LIN {X 0,Y 424.054,Z 656.663,A -85,B 0,C 180,E1 -10150.074,E2 -10150.074} C_VEL
LIN {X 0,Y 423.533,Z 671.263,A -85,B 0,C 180,E1 -10150.522,E2 -10150.522} C_VEL
LIN {X 0,Y 422.762,Z 685.237,A -85,B 0,C 180,E1 -10151.147,E2 -10151.147} C_VEL
LIN {X 0,Y 421.965,Z 698.713,A -85,B 0,C 180,E1 -10151.958,E2 -10151.958} C_VEL
LIN {X 0,Y 421.198,Z 710.972,A -85,B 0,C 180,E1 -10152.896,E2 -10152.896} C_VEL
LIN {X 0,Y 420.222,Z 722.559,A -85,B 0,C 180,E1 -10153.98,E2 -10153.98} C_VEL
LIN {X 0,Y 419.425,Z 733.214,A -85,B 0,C 180,E1 -10155.194,E2 -10155.194} C_VEL
LIN {X 0,Y 418.716,Z 743.545,A -85,B 0,C 180,E1 -10156.615,E2 -10156.615} C_VEL
LIN {X 0,Y 418.152,Z 752.53,A -85,B 0,C 180,E1 -10158.117,E2 -10158.117} C_VEL
LIN {X 0,Y 417.62,Z 760.846,A -85,B 0,C 180,E1 -10159.821,E2 -10159.821} C_VEL
LIN {X 0,Y 417.346,Z 766.695,A -85,B 0,C 180,E1 -10161.282,E2 -10161.282} C_VEL
LIN {X 0,Y 417.226,Z 772.808,A -85,B 0,C 180,E1 -10163.227,E2 -10163.227} C_VEL
LIN {X 0,Y 417.146,Z 777.257,A -85,B 0,C 180,E1 -10165.167,E2 -10165.167} C_VEL
LIN {X 0,Y 417.168,Z 780.178,A -85,B 0,C 180,E1 -10167.102,E2 -10167.102} C_VEL
LIN {X 0,Y 417.105,Z 781.632,A -85,B 0,C 180,E1 -10169.033,E2 -10169.033} C_VEL
LIN {X 0,Y 417.104,Z 781.632,A -85,B 0,C 180,E1 -10170.964,E2 -10170.964} C_VEL
LIN {X 0,Y 417.168,Z 780.18,A -85,B 0,C 180,E1 -10172.896,E2 -10172.896} C_VEL
LIN {X 0,Y 417.145,Z 777.26,A -85,B 0,C 180,E1 -10174.831,E2 -10174.831} C_VEL
LIN {X 0,Y 417.224,Z 772.806,A -85,B 0,C 180,E1 -10176.77,E2 -10176.77} C_VEL
LIN {X 0,Y 417.343,Z 766.691,A -85,B 0,C 180,E1 -10178.716,E2 -10178.716} C_VEL
LIN {X 0,Y 417.69,Z 759.788,A -85,B 0,C 180,E1 -10180.42,E2 -10180.42} C_VEL
LIN {X 0,Y 418.216,Z 751.155,A -85,B 0,C 180,E1 -10182.124,E2 -10182.124} C_VEL
LIN {X 0,Y 418.786,Z 742.137,A -85,B 0,C 180,E1 -10183.587,E2 -10183.587} C_VEL
LIN {X 0,Y 419.524,Z 731.202,A -85,B 0,C 180,E1 -10185.049,E2 -10185.049} C_VEL
LIN {X 0,Y 420.408,Z 720.153,A -85,B 0,C 180,E1 -10186.259,E2 -10186.259} C_VEL
LIN {X 0,Y 421.316,Z 708.059,A -85,B 0,C 180,E1 -10187.346,E2 -10187.346} C_VEL
LIN {X 0,Y 422.166,Z 695.251,A -85,B 0,C 180,E1 -10188.272,E2 -10188.272} C_VEL
LIN {X 0,Y 422.92,Z 682.408,A -85,B 0,C 180,E1 -10188.994,E2 -10188.994} C_VEL
LIN {X 0,Y 423.625,Z 667.816,A -85,B 0,C 180,E1 -10189.597,E2 -10189.597} C_VEL
LIN {X 0,Y 424.186,Z 653.721,A -85,B 0,C 180,E1 -10189.98,E2 -10189.98} C_VEL
LIN {X 0,Y 425.832,Z 546.42,A -85,B 0,C 180,E1 -10191.936,E2 -10191.936} C_VEL
LIN {X 0,Y 422.287,Z 522.478,A -85,B 0,C 180,E1 -10192.569,E2 -10192.569} C_VEL
LIN {X 0,Y 424.11,Z 501.54,A -85,B 0,C 180,E1 -10195.783,E2 -10195.783} C_VEL
LIN {X 0,Y 424.559,Z 496.002,A -85,B 0,C 180,E1 -10196.633,E2 -10196.633} C_VEL
LIN {X 0,Y 421.696,Z 483.135,A -85,B 0,C 180,E1 -10198.9,E2 -10198.9} C_VEL
LIN {X 0,Y 418.25,Z 470.012,A -85,B 0,C 180,E1 -10201.362,E2 -10201.362} C_VEL
LIN {X 0,Y 418.254,Z 469.992,A -85,B 0,C 180,E1 -10204.84,E2 -10204.84} C_VEL
LIN {X 0,Y 418.261,Z 470.007,A -85,B 0,C 180,E1 -10208.439,E2 -10208.439} C_VEL
LIN {X 0,Y 418.285,Z 470.007,A -85,B 0,C 180,E1 -10212.225,E2 -10212.225} C_VEL
LIN {X 0,Y 418.266,Z 470.007,A -85,B 0,C 180,E1 -10215.113,E2 -10215.113} C_VEL
LIN {X 0,Y 418.284,Z 470.001,A -85,B 0,C 180,E1 -10217.772,E2 -10217.772} C_VEL
LIN {X 0,Y 418.258,Z 470.004,A -85,B 0,C 180,E1 -10221.559,E2 -10221.559} C_VEL
LIN {X 0,Y 418.25,Z 470.001,A -85,B 0,C 180,E1 -10225.158,E2 -10225.158} C_VEL
LIN {X 0,Y 418.239,Z 470.007,A -85,B 0,C 180,E1 -10227.471,E2 -10227.471} C_VEL
LIN {X 0,Y 418.267,Z 470.008,A -85,B 0,C 180,E1 -10230.892,E2 -10230.892} C_VEL
LIN {X 0,Y 418.261,Z 470.008,A -85,B 0,C 180,E1 -10234.095,E2 -10234.095} C_VEL
LIN {X 0,Y 418.227,Z 469.991,A -85,B 0,C 180,E1 -10237.263,E2 -10237.263} C_VEL
LIN {X 0,Y 418.272,Z 470.001,A -85,B 0,C 180,E1 -10240.364,E2 -10240.364} C_VEL
LIN {X 0,Y 418.305,Z 469.998,A -85,B 0,C 180,E1 -10243.404,E2 -10243.404} C_VEL
LIN {X 0,Y 418.344,Z 469.997,A -85,B 0,C 180,E1 -10246.993,E2 -10246.993} C_VEL
LIN {X 0,Y 418.35,Z 469.996,A -85,B 0,C 180,E1 -10250.329,E2 -10250.329} C_VEL
LIN {X 0,Y 418.483,Z 469.972,A -85,B 0,C 180,E1 -10253.249,E2 -10253.249} C_VEL
LIN {X 0,Y 418.334,Z 469.999,A -85,B 0,C 180,E1 -10255.182,E2 -10255.182} C_VEL
LIN {X 0,Y 418.534,Z 469.971,A -85,B 0,C 180,E1 -10258.076,E2 -10258.076} C_VEL
LIN {X 0,Y 418.663,Z 469.955,A -85,B 0,C 180,E1 -10260,E2 -10260} C_VEL
LIN {X 0,Y 418.501,Z 469.972,A -85,B 0,C 180,E1 -10262.888,E2 -10262.888} C_VEL
LIN {X 0,Y 418.482,Z 469.981,A -85,B 0,C 180,E1 -10266.751,E2 -10266.751} C_VEL
LIN {X 0,Y 418.349,Z 469.993,A -85,B 0,C 180,E1 -10269.671,E2 -10269.671} C_VEL
LIN {X 0,Y 418.344,Z 469.992,A -85,B 0,C 180,E1 -10273.007,E2 -10273.007} C_VEL
LIN {X 0,Y 418.309,Z 470.001,A -85,B 0,C 180,E1 -10276.74,E2 -10276.74} C_VEL
LIN {X 0,Y 418.26,Z 470.007,A -85,B 0,C 180,E1 -10279.791,E2 -10279.791} C_VEL
LIN {X 0,Y 418.228,Z 470.012,A -85,B 0,C 180,E1 -10282.737,E2 -10282.737} C_VEL
LIN {X 0,Y 418.261,Z 470.006,A -85,B 0,C 180,E1 -10285.905,E2 -10285.905} C_VEL
LIN {X 0,Y 418.265,Z 470.005,A -85,B 0,C 180,E1 -10289.162,E2 -10289.162} C_VEL
LIN {X 0,Y 418.252,Z 470.008,A -85,B 0,C 180,E1 -10292.846,E2 -10292.846} C_VEL
LIN {X 0,Y 418.241,Z 470.014,A -85,B 0,C 180,E1 -10296.24,E2 -10296.24} C_VEL
LIN {X 0,Y 418.259,Z 470.008,A -85,B 0,C 180,E1 -10299.681,E2 -10299.681} C_VEL
LIN {X 0,Y 418.238,Z 470.016,A -85,B 0,C 180,E1 -10302.325,E2 -10302.325} C_VEL
LIN {X 0,Y 418.252,Z 470.009,A -85,B 0,C 180,E1 -10305.113,E2 -10305.113} C_VEL
LIN {X 0,Y 418.287,Z 470.005,A -85,B 0,C 180,E1 -10307.775,E2 -10307.775} C_VEL
LIN {X 0,Y 418.262,Z 470.008,A -85,B 0,C 180,E1 -10311.561,E2 -10311.561} C_VEL
LIN {X 0,Y 418.256,Z 470.009,A -85,B 0,C 180,E1 -10315.161,E2 -10315.161} C_VEL
LIN {X 0,Y 418.246,Z 470.012,A -85,B 0,C 180,E1 -10317.474,E2 -10317.474} C_VEL
LIN {X 0,Y 418.307,Z 470.145,A -85,B 0,C 180,E1 -10321.02,E2 -10321.02} C_VEL
LIN {X 0,Y 420.841,Z 480.928,A -85,B 0,C 180,E1 -10323.468,E2 -10323.468} C_VEL
LIN {X 0,Y 422.602,Z 489.933,A -85,B 0,C 180,E1 -10325.435,E2 -10325.435} C_VEL
LIN {X 0,Y 422.061,Z 498.987,A -85,B 0,C 180,E1 -10327.224,E2 -10327.224} C_VEL
LIN {X 0,Y 420.862,Z 516.189,A -85,B 0,C 180,E1 -10330.519,E2 -10330.519} C_VEL
LIN {X 0,Y 425.15,Z 538.523,A -85,B 0,C 180,E1 -10331.115,E2 -10331.115} C_VEL
LIN {X 0,Y 424.311,Z 628.226,A -85,B 0,C 180,E1 -10332.531,E2 -10332.531} C_VEL
LIN {X 0,Y 424.007,Z 641.22,A -85,B 0,C 180,E1 -10332.922,E2 -10332.922} C_VEL
LIN {X 0,Y 423.4,Z 653.756,A -85,B 0,C 180,E1 -10333.487,E2 -10333.487} C_VEL
LIN {X 0,Y 422.814,Z 665.376,A -85,B 0,C 180,E1 -10334.207,E2 -10334.207} C_VEL
LIN {X 0,Y 422.07,Z 676.227,A -85,B 0,C 180,E1 -10335.071,E2 -10335.071} C_VEL
LIN {X 0,Y 421.183,Z 686.717,A -85,B 0,C 180,E1 -10336.123,E2 -10336.123} C_VEL
LIN {X 0,Y 420.405,Z 695.493,A -85,B 0,C 180,E1 -10337.204,E2 -10337.204} C_VEL
LIN {X 0,Y 419.674,Z 703.55,A -85,B 0,C 180,E1 -10338.409,E2 -10338.409} C_VEL
LIN {X 0,Y 419.008,Z 711.29,A -85,B 0,C 180,E1 -10339.827,E2 -10339.827} C_VEL
LIN {X 0,Y 418.046,Z 714.527,A -85,B 0,C 180,E1 -10340.493,E2 -10340.493} C_VEL
LIN {X 0,Y 414.737,Z 719.395,A -85,B 0,C 180,E1 -10341.593,E2 -10341.593} C_VEL
LIN {X 0,Y 411.509,Z 723.632,A -85,B 0,C 180,E1 -10342.755,E2 -10342.755} C_VEL
LIN {X 0,Y 410.683,Z 725.814,A -85,B 0,C 180,E1 -10343.508,E2 -10343.508} C_VEL
LIN {X 0,Y 410.351,Z 729.419,A -85,B 0,C 180,E1 -10345.089,E2 -10345.089} C_VEL
LIN {X 0,Y 410.376,Z 731.097,A -85,B 0,C 180,E1 -10346.073,E2 -10346.073} C_VEL
LIN {X 0,Y 410.123,Z 733.306,A -85,B 0,C 180,E1 -10348.037,E2 -10348.037} C_VEL
LIN {X 0,Y 410.036,Z 734.085,A -85,B 0,C 180,E1 -10350.001,E2 -10350.001} C_VEL
LIN {X 0,Y 410.123,Z 733.376,A -85,B 0,C 180,E1 -10351.965,E2 -10351.965} C_VEL
LIN {X 0,Y 410.348,Z 731.224,A -85,B 0,C 180,E1 -10353.93,E2 -10353.93} C_VEL
LIN {X 0,Y 410.365,Z 728.597,A -85,B 0,C 180,E1 -10355.406,E2 -10355.406} C_VEL
LIN {X 0,Y 410.824,Z 724.254,A -85,B 0,C 180,E1 -10357.154,E2 -10357.154} C_VEL
LIN {X 0,Y 411.293,Z 718.604,A -85,B 0,C 180,E1 -10358.848,E2 -10358.848} C_VEL
LIN {X 0,Y 411.95,Z 712.331,A -85,B 0,C 180,E1 -10360.32,E2 -10360.32} C_VEL
LIN {X 0,Y 412.735,Z 704.546,A -85,B 0,C 180,E1 -10361.792,E2 -10361.792} C_VEL
LIN {X 0,Y 413.469,Z 696.618,A -85,B 0,C 180,E1 -10363.017,E2 -10363.017} C_VEL
LIN {X 0,Y 414.396,Z 686.951,A -85,B 0,C 180,E1 -10364.237,E2 -10364.237} C_VEL
LIN {X 0,Y 415.199,Z 676.497,A -85,B 0,C 180,E1 -10365.304,E2 -10365.304} C_VEL
LIN {X 0,Y 416.029,Z 665.54,A -85,B 0,C 180,E1 -10366.186,E2 -10366.186} C_VEL
LIN {X 0,Y 416.738,Z 653.875,A -85,B 0,C 180,E1 -10366.914,E2 -10366.914} C_VEL
LIN {X 0,Y 417.301,Z 640.506,A -85,B 0,C 180,E1 -10367.521,E2 -10367.521} C_VEL
LIN {X 0,Y 417.704,Z 628.087,A -85,B 0,C 180,E1 -10367.883,E2 -10367.883} C_VEL
LIN {X 0,Y 418.405,Z 538.602,A -85,B 0,C 180,E1 -10369.325,E2 -10369.325} C_VEL
LIN {X 0,Y 414.057,Z 516.251,A -85,B 0,C 180,E1 -10369.943,E2 -10369.943} C_VEL
LIN {X 0,Y 415.253,Z 499.637,A -85,B 0,C 180,E1 -10373.173,E2 -10373.173} C_VEL
LIN {X 0,Y 415.804,Z 491.874,A -85,B 0,C 180,E1 -10374.73,E2 -10374.73} C_VEL
LIN {X 0,Y 413.438,Z 480.243,A -85,B 0,C 180,E1 -10377.322,E2 -10377.322} C_VEL
LIN {X 0,Y 411.221,Z 470.895,A -85,B 0,C 180,E1 -10379.542,E2 -10379.542} C_VEL
LIN {X 0,Y 411.212,Z 470.889,A -85,B 0,C 180,E1 -10383.156,E2 -10383.156} C_VEL
LIN {X 0,Y 411.201,Z 470.887,A -85,B 0,C 180,E1 -10386.554,E2 -10386.554} C_VEL
LIN {X 0,Y 411.225,Z 470.89,A -85,B 0,C 180,E1 -10389.729,E2 -10389.729} C_VEL
LIN {X 0,Y 411.184,Z 470.892,A -85,B 0,C 180,E1 -10393.133,E2 -10393.133} C_VEL
LIN {X 0,Y 411.175,Z 470.895,A -85,B 0,C 180,E1 -10395.881,E2 -10395.881} C_VEL
LIN {X 0,Y 411.169,Z 470.888,A -85,B 0,C 180,E1 -10398.772,E2 -10398.772} C_VEL
LIN {X 0,Y 411.202,Z 470.881,A -85,B 0,C 180,E1 -10402.027,E2 -10402.027} C_VEL
LIN {X 0,Y 411.213,Z 470.89,A -85,B 0,C 180,E1 -10405.667,E2 -10405.667} C_VEL
LIN {X 0,Y 411.196,Z 470.89,A -85,B 0,C 180,E1 -10409.153,E2 -10409.153} C_VEL
LIN {X 0,Y 411.277,Z 471.015,A -85,B 0,C 180,E1 -10411.233,E2 -10411.233} C_VEL
LIN {X 0,Y 414.611,Z 486.116,A -85,B 0,C 180,E1 -10413.949,E2 -10413.949} C_VEL
LIN {X 0,Y 415.396,Z 491.985,A -85,B 0,C 180,E1 -10414.978,E2 -10414.978} C_VEL
LIN {X 0,Y 414.357,Z 514.361,A -85,B 0,C 180,E1 -10418.639,E2 -10418.639} C_VEL
LIN {X 0,Y 413.73,Z 529.022,A -85,B 0,C 180,E1 -10421.042,E2 -10421.042} C_VEL
LIN {X 0,Y 416.567,Z 548.221,A -85,B 0,C 180,E1 -10421.577,E2 -10421.577} C_VEL
LIN {X 0,Y 414.847,Z 640.02,A -85,B 0,C 180,E1 -10423.483,E2 -10423.483} C_VEL
LIN {X 0,Y 414.531,Z 653.035,A -85,B 0,C 180,E1 -10423.945,E2 -10423.945} C_VEL
LIN {X 0,Y 414.003,Z 666.156,A -85,B 0,C 180,E1 -10424.618,E2 -10424.618} C_VEL
LIN {X 0,Y 413.427,Z 678.373,A -85,B 0,C 180,E1 -10425.456,E2 -10425.456} C_VEL
LIN {X 0,Y 412.841,Z 689.793,A -85,B 0,C 180,E1 -10426.463,E2 -10426.463} C_VEL
LIN {X 0,Y 412.207,Z 699.947,A -85,B 0,C 180,E1 -10427.57,E2 -10427.57} C_VEL
LIN {X 0,Y 411.644,Z 709.929,A -85,B 0,C 180,E1 -10428.926,E2 -10428.926} C_VEL
LIN {X 0,Y 411.121,Z 718.723,A -85,B 0,C 180,E1 -10430.405,E2 -10430.405} C_VEL
LIN {X 0,Y 410.693,Z 725.71,A -85,B 0,C 180,E1 -10431.884,E2 -10431.884} C_VEL
LIN {X 0,Y 410.378,Z 732.281,A -85,B 0,C 180,E1 -10433.66,E2 -10433.66} C_VEL
LIN {X 0,Y 410.196,Z 736.265,A -85,B 0,C 180,E1 -10435.085,E2 -10435.085} C_VEL
LIN {X 0,Y 410.125,Z 738.391,A -85,B 0,C 180,E1 -10436.069,E2 -10436.069} C_VEL
LIN {X 0,Y 410.143,Z 740.08,A -85,B 0,C 180,E1 -10437.053,E2 -10437.053} C_VEL
LIN {X 0,Y 410.053,Z 741.351,A -85,B 0,C 180,E1 -10438.035,E2 -10438.035} C_VEL
LIN {X 0,Y 409.984,Z 742.151,A -85,B 0,C 180,E1 -10439.018,E2 -10439.018} C_VEL
LIN {X 0,Y 409.973,Z 742.541,A -85,B 0,C 180,E1 -10440,E2 -10440} C_VEL
LIN {X 0,Y 410.007,Z 742.527,A -85,B 0,C 180,E1 -10440.982,E2 -10440.982} C_VEL
LIN {X 0,Y 410.072,Z 742.051,A -85,B 0,C 180,E1 -10441.964,E2 -10441.964} C_VEL
LIN {X 0,Y 410.184,Z 741.151,A -85,B 0,C 180,E1 -10442.946,E2 -10442.946} C_VEL
LIN {X 0,Y 410.305,Z 739.842,A -85,B 0,C 180,E1 -10443.929,E2 -10443.929} C_VEL
LIN {X 0,Y 410.31,Z 737.029,A -85,B 0,C 180,E1 -10445.406,E2 -10445.406} C_VEL
LIN {X 0,Y 410.673,Z 732.811,A -85,B 0,C 180,E1 -10446.98,E2 -10446.98} C_VEL
LIN {X 0,Y 411.022,Z 727.012,A -85,B 0,C 180,E1 -10448.604,E2 -10448.604} C_VEL
LIN {X 0,Y 411.6,Z 720.3,A -85,B 0,C 180,E1 -10450.08,E2 -10450.08} C_VEL
LIN {X 0,Y 412.186,Z 711.938,A -85,B 0,C 180,E1 -10451.557,E2 -10451.557} C_VEL
LIN {X 0,Y 412.774,Z 703.343,A -85,B 0,C 180,E1 -10452.788,E2 -10452.788} C_VEL
LIN {X 0,Y 413.525,Z 693.729,A -85,B 0,C 180,E1 -10453.911,E2 -10453.911} C_VEL
LIN {X 0,Y 414.23,Z 683.684,A -85,B 0,C 180,E1 -10454.869,E2 -10454.869} C_VEL
LIN {X 0,Y 414.808,Z 672.46,A -85,B 0,C 180,E1 -10455.729,E2 -10455.729} C_VEL
LIN {X 0,Y 415.449,Z 660.062,A -85,B 0,C 180,E1 -10456.46,E2 -10456.46} C_VEL
LIN {X 0,Y 415.999,Z 646.362,A -85,B 0,C 180,E1 -10457.038,E2 -10457.038} C_VEL
LIN {X 0,Y 416.385,Z 633.029,A -85,B 0,C 180,E1 -10457.402,E2 -10457.402} C_VEL
LIN {X 0,Y 418.682,Z 549.557,A -85,B 0,C 180,E1 -10459.31,E2 -10459.31} C_VEL
LIN {X 0,Y 418.156,Z 544.537,A -85,B 0,C 180,E1 -10459.475,E2 -10459.475} C_VEL
LIN {X 0,Y 415.628,Z 531.798,A -85,B 0,C 180,E1 -10460.024,E2 -10460.024} C_VEL
LIN {X 0,Y 416.725,Z 509.735,A -85,B 0,C 180,E1 -10463.612,E2 -10463.612} C_VEL
LIN {X 0,Y 417.52,Z 495.37,A -85,B 0,C 180,E1 -10465.954,E2 -10465.954} C_VEL
LIN {X 0,Y 416.207,Z 487.66,A -85,B 0,C 180,E1 -10467.346,E2 -10467.346} C_VEL
LIN {X 0,Y 413.733,Z 478.663,A -85,B 0,C 180,E1 -10469.119,E2 -10469.119} C_VEL
LIN {X 0,Y 411.206,Z 470.894,A -85,B 0,C 180,E1 -10470.775,E2 -10470.775} C_VEL
LIN {X 0,Y 411.211,Z 470.889,A -85,B 0,C 180,E1 -10474.333,E2 -10474.333} C_VEL
LIN {X 0,Y 411.206,Z 470.891,A -85,B 0,C 180,E1 -10477.972,E2 -10477.972} C_VEL
LIN {X 0,Y 411.188,Z 470.89,A -85,B 0,C 180,E1 -10480.503,E2 -10480.503} C_VEL
LIN {X 0,Y 411.178,Z 470.893,A -85,B 0,C 180,E1 -10483.133,E2 -10483.133} C_VEL
LIN {X 0,Y 411.173,Z 470.893,A -85,B 0,C 180,E1 -10485.88,E2 -10485.88} C_VEL
LIN {X 0,Y 411.168,Z 470.891,A -85,B 0,C 180,E1 -10488.771,E2 -10488.771} C_VEL
LIN {X 0,Y 411.196,Z 470.889,A -85,B 0,C 180,E1 -10492.025,E2 -10492.025} C_VEL
LIN {X 0,Y 411.21,Z 470.888,A -85,B 0,C 180,E1 -10495.666,E2 -10495.666} C_VEL
LIN {X 0,Y 411.206,Z 471.062,A -85,B 0,C 180,E1 -10498.248,E2 -10498.248} C_VEL
LIN {X 0,Y 414.819,Z 484.656,A -85,B 0,C 180,E1 -10500.848,E2 -10500.848} C_VEL
LIN {X 0,Y 417.698,Z 497.09,A -85,B 0,C 180,E1 -10503.095,E2 -10503.095} C_VEL
LIN {X 0,Y 416.577,Z 511.136,A -85,B 0,C 180,E1 -10505.296,E2 -10505.296} C_VEL
LIN {X 0,Y 415.53,Z 522.528,A -85,B 0,C 180,E1 -10507.073,E2 -10507.073} C_VEL
LIN {X 0,Y 419.162,Z 546.888,A -85,B 0,C 180,E1 -10507.727,E2 -10507.727} C_VEL
LIN {X 0,Y 417.606,Z 646.176,A -85,B 0,C 180,E1 -10509.56,E2 -10509.56} C_VEL
LIN {X 0,Y 417.135,Z 662.283,A -85,B 0,C 180,E1 -10509.922,E2 -10509.922} C_VEL
LIN {X 0,Y 416.552,Z 675.692,A -85,B 0,C 180,E1 -10510.406,E2 -10510.406} C_VEL
LIN {X 0,Y 415.783,Z 689.015,A -85,B 0,C 180,E1 -10511.074,E2 -10511.074} C_VEL
LIN {X 0,Y 414.919,Z 701.982,A -85,B 0,C 180,E1 -10511.928,E2 -10511.928} C_VEL
LIN {X 0,Y 413.997,Z 714.542,A -85,B 0,C 180,E1 -10512.971,E2 -10512.971} C_VEL
LIN {X 0,Y 413.081,Z 725.442,A -85,B 0,C 180,E1 -10514.076,E2 -10514.076} C_VEL
LIN {X 0,Y 412.206,Z 736.464,A -85,B 0,C 180,E1 -10515.434,E2 -10515.434} C_VEL
LIN {X 0,Y 411.429,Z 746.705,A -85,B 0,C 180,E1 -10516.968,E2 -10516.968} C_VEL
LIN {X 0,Y 410.893,Z 755.881,A -85,B 0,C 180,E1 -10518.655,E2 -10518.655} C_VEL
LIN {X 0,Y 410.479,Z 762.498,A -85,B 0,C 180,E1 -10520.14,E2 -10520.14} C_VEL
LIN {X 0,Y 410.231,Z 767.948,A -85,B 0,C 180,E1 -10521.626,E2 -10521.626} C_VEL
LIN {X 0,Y 410.137,Z 772.384,A -85,B 0,C 180,E1 -10523.11,E2 -10523.11} C_VEL
LIN {X 0,Y 410.077,Z 776.842,A -85,B 0,C 180,E1 -10525.083,E2 -10525.083} C_VEL
LIN {X 0,Y 410.066,Z 779.765,A -85,B 0,C 180,E1 -10527.052,E2 -10527.052} C_VEL
LIN {X 0,Y 410.025,Z 781.223,A -85,B 0,C 180,E1 -10529.017,E2 -10529.017} C_VEL
LIN {X 0,Y 410.024,Z 781.223,A -85,B 0,C 180,E1 -10530.981,E2 -10530.981} C_VEL
LIN {X 0,Y 410.065,Z 779.767,A -85,B 0,C 180,E1 -10532.946,E2 -10532.946} C_VEL
LIN {X 0,Y 410.076,Z 776.844,A -85,B 0,C 180,E1 -10534.914,E2 -10534.914} C_VEL
LIN {X 0,Y 410.135,Z 772.381,A -85,B 0,C 180,E1 -10536.888,E2 -10536.888} C_VEL
LIN {X 0,Y 410.286,Z 766.258,A -85,B 0,C 180,E1 -10538.867,E2 -10538.867} C_VEL
LIN {X 0,Y 410.637,Z 759.34,A -85,B 0,C 180,E1 -10540.601,E2 -10540.601} C_VEL
LIN {X 0,Y 411.111,Z 752.065,A -85,B 0,C 180,E1 -10542.087,E2 -10542.087} C_VEL
LIN {X 0,Y 411.696,Z 743.519,A -85,B 0,C 180,E1 -10543.542,E2 -10543.542} C_VEL
LIN {X 0,Y 412.354,Z 734.623,A -85,B 0,C 180,E1 -10544.811,E2 -10544.811} C_VEL
LIN {X 0,Y 413.157,Z 724.329,A -85,B 0,C 180,E1 -10546.045,E2 -10546.045} C_VEL
LIN {X 0,Y 414.061,Z 713.205,A -85,B 0,C 180,E1 -10547.151,E2 -10547.151} C_VEL
LIN {X 0,Y 414.982,Z 700.577,A -85,B 0,C 180,E1 -10548.173,E2 -10548.173} C_VEL
LIN {X 0,Y 415.883,Z 686.726,A -85,B 0,C 180,E1 -10549.047,E2 -10549.047} C_VEL
LIN {X 0,Y 416.657,Z 672.603,A -85,B 0,C 180,E1 -10549.714,E2 -10549.714} C_VEL
LIN {X 0,Y 417.28,Z 658.88,A -85,B 0,C 180,E1 -10550.165,E2 -10550.165} C_VEL
LIN {X 0,Y 417.961,Z 627.698,A -85,B 0,C 180,E1 -10550.773,E2 -10550.773} C_VEL
LIN {X 0,Y 419.118,Z 546.764,A -85,B 0,C 180,E1 -10552.27,E2 -10552.27} C_VEL
LIN {X 0,Y 415.522,Z 522.441,A -85,B 0,C 180,E1 -10552.924,E2 -10552.924} C_VEL
LIN {X 0,Y 417.442,Z 501.494,A -85,B 0,C 180,E1 -10556.2,E2 -10556.2} C_VEL
LIN {X 0,Y 417.667,Z 497.09,A -85,B 0,C 180,E1 -10556.897,E2 -10556.897} C_VEL
LIN {X 0,Y 414.387,Z 482.95,A -85,B 0,C 180,E1 -10559.46,E2 -10559.46} C_VEL
LIN {X 0,Y 411.185,Z 470.892,A -85,B 0,C 180,E1 -10561.798,E2 -10561.798} C_VEL
LIN {X 0,Y 411.206,Z 470.87,A -85,B 0,C 180,E1 -10564.877,E2 -10564.877} C_VEL
LIN {X 0,Y 411.21,Z 470.886,A -85,B 0,C 180,E1 -10568.169,E2 -10568.169} C_VEL
LIN {X 0,Y 411.203,Z 470.889,A -85,B 0,C 180,E1 -10571.235,E2 -10571.235} C_VEL
LIN {X 0,Y 411.225,Z 470.887,A -85,B 0,C 180,E1 -10574.481,E2 -10574.481} C_VEL
LIN {X 0,Y 411.224,Z 470.882,A -85,B 0,C 180,E1 -10577.295,E2 -10577.295} C_VEL
LIN {X 0,Y 411.223,Z 470.884,A -85,B 0,C 180,E1 -10580.777,E2 -10580.777} C_VEL
LIN {X 0,Y 411.19,Z 470.872,A -85,B 0,C 180,E1 -10584.471,E2 -10584.471} C_VEL
LIN {X 0,Y 411.162,Z 470.889,A -85,B 0,C 180,E1 -10588.002,E2 -10588.002} C_VEL
LIN {X 0,Y 411.214,Z 470.882,A -85,B 0,C 180,E1 -10591.41,E2 -10591.41} C_VEL
LIN {X 0,Y 411.226,Z 470.886,A -85,B 0,C 180,E1 -10594.706,E2 -10594.706} C_VEL
LIN {X 0,Y 411.194,Z 470.865,A -85,B 0,C 180,E1 -10597.913,E2 -10597.913} C_VEL
LIN {X 0,Y 411.214,Z 470.887,A -85,B 0,C 180,E1 -10601.051,E2 -10601.051} C_VEL
LIN {X 0,Y 411.244,Z 470.879,A -85,B 0,C 180,E1 -10604.131,E2 -10604.131} C_VEL
LIN {X 0,Y 411.304,Z 470.873,A -85,B 0,C 180,E1 -10607.166,E2 -10607.166} C_VEL
LIN {X 0,Y 411.298,Z 470.873,A -85,B 0,C 180,E1 -10610.161,E2 -10610.161} C_VEL
LIN {X 0,Y 411.45,Z 470.848,A -85,B 0,C 180,E1 -10613.133,E2 -10613.133} C_VEL
LIN {X 0,Y 411.304,Z 470.875,A -85,B 0,C 180,E1 -10615.099,E2 -10615.099} C_VEL
LIN {X 0,Y 411.503,Z 470.847,A -85,B 0,C 180,E1 -10618.043,E2 -10618.043} C_VEL
LIN {X 0,Y 411.633,Z 470.831,A -85,B 0,C 180,E1 -10620,E2 -10620} C_VEL
LIN {X 0,Y 411.456,Z 470.849,A -85,B 0,C 180,E1 -10622.937,E2 -10622.937} C_VEL
LIN {X 0,Y 411.449,Z 470.856,A -85,B 0,C 180,E1 -10626.867,E2 -10626.867} C_VEL
LIN {X 0,Y 411.298,Z 470.872,A -85,B 0,C 180,E1 -10629.839,E2 -10629.839} C_VEL
LIN {X 0,Y 411.302,Z 470.868,A -85,B 0,C 180,E1 -10633.11,E2 -10633.11} C_VEL
LIN {X 0,Y 411.253,Z 470.878,A -85,B 0,C 180,E1 -10636.87,E2 -10636.87} C_VEL
LIN {X 0,Y 411.22,Z 470.885,A -85,B 0,C 180,E1 -10639.988,E2 -10639.988} C_VEL
LIN {X 0,Y 411.193,Z 470.887,A -85,B 0,C 180,E1 -10643.148,E2 -10643.148} C_VEL
LIN {X 0,Y 411.228,Z 470.882,A -85,B 0,C 180,E1 -10646.382,E2 -10646.382} C_VEL
LIN {X 0,Y 411.202,Z 470.884,A -85,B 0,C 180,E1 -10649.713,E2 -10649.713} C_VEL
LIN {X 0,Y 411.198,Z 470.884,A -85,B 0,C 180,E1 -10653.157,E2 -10653.157} C_VEL
LIN {X 0,Y 411.188,Z 470.89,A -85,B 0,C 180,E1 -10656.554,E2 -10656.554} C_VEL
LIN {X 0,Y 411.221,Z 470.885,A -85,B 0,C 180,E1 -10659.732,E2 -10659.732} C_VEL
LIN {X 0,Y 411.17,Z 470.891,A -85,B 0,C 180,E1 -10663.134,E2 -10663.134} C_VEL
LIN {X 0,Y 411.23,Z 470.884,A -85,B 0,C 180,E1 -10665.873,E2 -10665.873} C_VEL
LIN {X 0,Y 411.205,Z 470.891,A -85,B 0,C 180,E1 -10668.766,E2 -10668.766} C_VEL
LIN {X 0,Y 411.201,Z 470.888,A -85,B 0,C 180,E1 -10672.029,E2 -10672.029} C_VEL
LIN {X 0,Y 411.203,Z 470.886,A -85,B 0,C 180,E1 -10675.668,E2 -10675.668} C_VEL
LIN {X 0,Y 411.197,Z 470.887,A -85,B 0,C 180,E1 -10679.155,E2 -10679.155} C_VEL
LIN {X 0,Y 411.239,Z 471.069,A -85,B 0,C 180,E1 -10680.643,E2 -10680.643} C_VEL
LIN {X 0,Y 413.945,Z 482.371,A -85,B 0,C 180,E1 -10683.263,E2 -10683.263} C_VEL
LIN {X 0,Y 415.722,Z 491.396,A -85,B 0,C 180,E1 -10685.268,E2 -10685.268} C_VEL
LIN {X 0,Y 415.322,Z 499.161,A -85,B 0,C 180,E1 -10686.833,E2 -10686.833} C_VEL
LIN {X 0,Y 414.019,Z 516.251,A -85,B 0,C 180,E1 -10690.155,E2 -10690.155} C_VEL
LIN {X 0,Y 418.491,Z 539.512,A -85,B 0,C 180,E1 -10690.79,E2 -10690.79} C_VEL
LIN {X 0,Y 417.605,Z 629.408,A -85,B 0,C 180,E1 -10692.241,E2 -10692.241} C_VEL
LIN {X 0,Y 417.204,Z 642.861,A -85,B 0,C 180,E1 -10692.667,E2 -10692.667} C_VEL
LIN {X 0,Y 416.557,Z 655.602,A -85,B 0,C 180,E1 -10693.271,E2 -10693.271} C_VEL
LIN {X 0,Y 415.871,Z 667.636,A -85,B 0,C 180,E1 -10694.062,E2 -10694.062} C_VEL
LIN {X 0,Y 415.076,Z 678.578,A -85,B 0,C 180,E1 -10694.991,E2 -10694.991} C_VEL
LIN {X 0,Y 414.134,Z 689.316,A -85,B 0,C 180,E1 -10696.132,E2 -10696.132} C_VEL
LIN {X 0,Y 413.337,Z 697.709,A -85,B 0,C 180,E1 -10697.231,E2 -10697.231} C_VEL
LIN {X 0,Y 412.6,Z 705.451,A -85,B 0,C 180,E1 -10698.456,E2 -10698.456} C_VEL
LIN {X 0,Y 411.909,Z 713.07,A -85,B 0,C 180,E1 -10699.929,E2 -10699.929} C_VEL
LIN {X 0,Y 411.309,Z 718.242,A -85,B 0,C 180,E1 -10701.155,E2 -10701.155} C_VEL
LIN {X 0,Y 410.802,Z 724.059,A -85,B 0,C 180,E1 -10702.871,E2 -10702.871} C_VEL
LIN {X 0,Y 410.683,Z 725.814,A -85,B 0,C 180,E1 -10703.508,E2 -10703.508} C_VEL
LIN {X 0,Y 409.896,Z 727.804,A -85,B 0,C 180,E1 -10704.277,E2 -10704.277} C_VEL
LIN {X 0,Y 406.861,Z 730.515,A -85,B 0,C 180,E1 -10705.546,E2 -10705.546} C_VEL
LIN {X 0,Y 404.319,Z 732.237,A -85,B 0,C 180,E1 -10706.589,E2 -10706.589} C_VEL
LIN {X 0,Y 403.118,Z 733.363,A -85,B 0,C 180,E1 -10707.545,E2 -10707.545} C_VEL
LIN {X 0,Y 403.081,Z 733.422,A -85,B 0,C 180,E1 -10707.684,E2 -10707.684} C_VEL
LIN {X 0,Y 402.967,Z 734.282,A -85,B 0,C 180,E1 -10709.002,E2 -10709.002} C_VEL
LIN {X 0,Y 402.967,Z 734.323,A -85,B 0,C 180,E1 -10711.001,E2 -10711.001} C_VEL
LIN {X 0,Y 403.179,Z 732.889,A -85,B 0,C 180,E1 -10712.999,E2 -10712.999} C_VEL
LIN {X 0,Y 403.276,Z 731.635,A -85,B 0,C 180,E1 -10713.999,E2 -10713.999} C_VEL
LIN {X 0,Y 403.318,Z 729.011,A -85,B 0,C 180,E1 -10715.501,E2 -10715.501} C_VEL
LIN {X 0,Y 403.752,Z 724.983,A -85,B 0,C 180,E1 -10717.166,E2 -10717.166} C_VEL
LIN {X 0,Y 404.301,Z 719.034,A -85,B 0,C 180,E1 -10719.002,E2 -10719.002} C_VEL
LIN {X 0,Y 404.99,Z 712.771,A -85,B 0,C 180,E1 -10720.5,E2 -10720.5} C_VEL
LIN {X 0,Y 405.792,Z 704.999,A -85,B 0,C 180,E1 -10721.996,E2 -10721.996} C_VEL
LIN {X 0,Y 406.584,Z 697.087,A -85,B 0,C 180,E1 -10723.241,E2 -10723.241} C_VEL
LIN {X 0,Y 407.552,Z 687.443,A -85,B 0,C 180,E1 -10724.481,E2 -10724.481} C_VEL
LIN {X 0,Y 408.415,Z 676.421,A -85,B 0,C 180,E1 -10725.622,E2 -10725.622} C_VEL
LIN {X 0,Y 409.248,Z 666.14,A -85,B 0,C 180,E1 -10726.462,E2 -10726.462} C_VEL
LIN {X 0,Y 410.002,Z 654.559,A -85,B 0,C 180,E1 -10727.2,E2 -10727.2} C_VEL
LIN {X 0,Y 410.581,Z 641.335,A -85,B 0,C 180,E1 -10727.818,E2 -10727.818} C_VEL
LIN {X 0,Y 411.019,Z 627.932,A -85,B 0,C 180,E1 -10728.217,E2 -10728.217} C_VEL
LIN {X 0,Y 411.804,Z 539.67,A -85,B 0,C 180,E1 -10729.658,E2 -10729.658} C_VEL
LIN {X 0,Y 407.234,Z 516.284,A -85,B 0,C 180,E1 -10730.324,E2 -10730.324} C_VEL
LIN {X 0,Y 408.4,Z 501.107,A -85,B 0,C 180,E1 -10733.317,E2 -10733.317} C_VEL
LIN {X 0,Y 408.924,Z 493.326,A -85,B 0,C 180,E1 -10734.903,E2 -10734.903} C_VEL
LIN {X 0,Y 406.262,Z 480.39,A -85,B 0,C 180,E1 -10737.846,E2 -10737.846} C_VEL
LIN {X 0,Y 404.164,Z 471.773,A -85,B 0,C 180,E1 -10739.899,E2 -10739.899} C_VEL
LIN {X 0,Y 404.177,Z 471.767,A -85,B 0,C 180,E1 -10743.421,E2 -10743.421} C_VEL
LIN {X 0,Y 404.15,Z 471.765,A -85,B 0,C 180,E1 -10746.247,E2 -10746.247} C_VEL
LIN {X 0,Y 404.165,Z 471.761,A -85,B 0,C 180,E1 -10748.757,E2 -10748.757} C_VEL
LIN {X 0,Y 404.131,Z 471.768,A -85,B 0,C 180,E1 -10751.601,E2 -10751.601} C_VEL
LIN {X 0,Y 404.155,Z 471.761,A -85,B 0,C 180,E1 -10754.523,E2 -10754.523} C_VEL
LIN {X 0,Y 404.142,Z 471.766,A -85,B 0,C 180,E1 -10757.296,E2 -10757.296} C_VEL
LIN {X 0,Y 404.175,Z 471.765,A -85,B 0,C 180,E1 -10759.956,E2 -10759.956} C_VEL
LIN {X 0,Y 404.145,Z 471.762,A -85,B 0,C 180,E1 -10763.125,E2 -10763.125} C_VEL
LIN {X 0,Y 404.152,Z 471.767,A -85,B 0,C 180,E1 -10766.188,E2 -10766.188} C_VEL
LIN {X 0,Y 404.152,Z 471.77,A -85,B 0,C 180,E1 -10769.715,E2 -10769.715} C_VEL
LIN {X 0,Y 404.235,Z 471.962,A -85,B 0,C 180,E1 -10770.976,E2 -10770.976} C_VEL
LIN {X 0,Y 407.569,Z 487.059,A -85,B 0,C 180,E1 -10773.726,E2 -10773.726} C_VEL
LIN {X 0,Y 408.498,Z 493.132,A -85,B 0,C 180,E1 -10774.798,E2 -10774.798} C_VEL
LIN {X 0,Y 407.463,Z 514.194,A -85,B 0,C 180,E1 -10778.286,E2 -10778.286} C_VEL
LIN {X 0,Y 406.832,Z 529.29,A -85,B 0,C 180,E1 -10780.773,E2 -10780.773} C_VEL
LIN {X 0,Y 409.735,Z 548.735,A -85,B 0,C 180,E1 -10781.324,E2 -10781.324} C_VEL
LIN {X 0,Y 407.908,Z 640.517,A -85,B 0,C 180,E1 -10783.291,E2 -10783.291} C_VEL
LIN {X 0,Y 407.617,Z 652.714,A -85,B 0,C 180,E1 -10783.729,E2 -10783.729} C_VEL
LIN {X 0,Y 407.05,Z 665.949,A -85,B 0,C 180,E1 -10784.413,E2 -10784.413} C_VEL
LIN {X 0,Y 406.469,Z 677.886,A -85,B 0,C 180,E1 -10785.232,E2 -10785.232} C_VEL
LIN {X 0,Y 405.904,Z 689.157,A -85,B 0,C 180,E1 -10786.227,E2 -10786.227} C_VEL
LIN {X 0,Y 405.266,Z 699.476,A -85,B 0,C 180,E1 -10787.353,E2 -10787.353} C_VEL
LIN {X 0,Y 404.726,Z 707.98,A -85,B 0,C 180,E1 -10788.481,E2 -10788.481} C_VEL
LIN {X 0,Y 404.181,Z 717.193,A -85,B 0,C 180,E1 -10789.986,E2 -10789.986} C_VEL
LIN {X 0,Y 403.708,Z 724.6,A -85,B 0,C 180,E1 -10791.49,E2 -10791.49} C_VEL
LIN {X 0,Y 403.387,Z 731.386,A -85,B 0,C 180,E1 -10793.262,E2 -10793.262} C_VEL
LIN {X 0,Y 403.138,Z 736.398,A -85,B 0,C 180,E1 -10794.999,E2 -10794.999} C_VEL
LIN {X 0,Y 403.036,Z 738.583,A -85,B 0,C 180,E1 -10796,E2 -10796} C_VEL
LIN {X 0,Y 403.047,Z 740.304,A -85,B 0,C 180,E1 -10797.001,E2 -10797.001} C_VEL
LIN {X 0,Y 402.985,Z 741.617,A -85,B 0,C 180,E1 -10798.001,E2 -10798.001} C_VEL
LIN {X 0,Y 402.909,Z 742.46,A -85,B 0,C 180,E1 -10799,E2 -10799} C_VEL
LIN {X 0,Y 402.895,Z 742.878,A -85,B 0,C 180,E1 -10800,E2 -10800} C_VEL
LIN {X 0,Y 402.931,Z 742.89,A -85,B 0,C 180,E1 -10800.999,E2 -10800.999} C_VEL
LIN {X 0,Y 403.004,Z 742.455,A -85,B 0,C 180,E1 -10801.999,E2 -10801.999} C_VEL
LIN {X 0,Y 403.126,Z 741.574,A -85,B 0,C 180,E1 -10802.998,E2 -10802.998} C_VEL
LIN {X 0,Y 403.23,Z 740.284,A -85,B 0,C 180,E1 -10803.998,E2 -10803.998} C_VEL
LIN {X 0,Y 403.269,Z 737.501,A -85,B 0,C 180,E1 -10805.5,E2 -10805.5} C_VEL
LIN {X 0,Y 403.63,Z 733.578,A -85,B 0,C 180,E1 -10807.024,E2 -10807.024} C_VEL
LIN {X 0,Y 403.953,Z 728.606,A -85,B 0,C 180,E1 -10808.504,E2 -10808.504} C_VEL
LIN {X 0,Y 404.546,Z 722.181,A -85,B 0,C 180,E1 -10810.004,E2 -10810.004} C_VEL
LIN {X 0,Y 405.141,Z 714.183,A -85,B 0,C 180,E1 -10811.507,E2 -10811.507} C_VEL
LIN {X 0,Y 405.777,Z 705.994,A -85,B 0,C 180,E1 -10812.758,E2 -10812.758} C_VEL
LIN {X 0,Y 406.59,Z 695.886,A -85,B 0,C 180,E1 -10814.004,E2 -10814.004} C_VEL
LIN {X 0,Y 407.439,Z 684.668,A -85,B 0,C 180,E1 -10815.123,E2 -10815.123} C_VEL
LIN {X 0,Y 408.077,Z 673.702,A -85,B 0,C 180,E1 -10815.995,E2 -10815.995} C_VEL
LIN {X 0,Y 408.772,Z 661.64,A -85,B 0,C 180,E1 -10816.737,E2 -10816.737} C_VEL
LIN {X 0,Y 409.331,Z 648.704,A -85,B 0,C 180,E1 -10817.324,E2 -10817.324} C_VEL
LIN {X 0,Y 409.782,Z 633.81,A -85,B 0,C 180,E1 -10817.756,E2 -10817.756} C_VEL
LIN {X 0,Y 411.759,Z 565.233,A -85,B 0,C 180,E1 -10819.369,E2 -10819.369} C_VEL
LIN {X 0,Y 412.229,Z 548.113,A -85,B 0,C 180,E1 -10819.799,E2 -10819.799} C_VEL
LIN {X 0,Y 409.45,Z 534.047,A -85,B 0,C 180,E1 -10820.392,E2 -10820.392} C_VEL
LIN {X 0,Y 409.074,Z 532.323,A -85,B 0,C 180,E1 -10820.49,E2 -10820.49} C_VEL
LIN {X 0,Y 410.263,Z 510.928,A -85,B 0,C 180,E1 -10824.007,E2 -10824.007} C_VEL
LIN {X 0,Y 411.01,Z 498.092,A -85,B 0,C 180,E1 -10826.123,E2 -10826.123} C_VEL
LIN {X 0,Y 410.097,Z 491.697,A -85,B 0,C 180,E1 -10827.321,E2 -10827.321} C_VEL
LIN {X 0,Y 407.855,Z 482.876,A -85,B 0,C 180,E1 -10829.077,E2 -10829.077} C_VEL
LIN {X 0,Y 404.143,Z 471.773,A -85,B 0,C 180,E1 -10831.504,E2 -10831.504} C_VEL
LIN {X 0,Y 404.191,Z 471.764,A -85,B 0,C 180,E1 -10835.015,E2 -10835.015} C_VEL
LIN {X 0,Y 404.164,Z 471.764,A -85,B 0,C 180,E1 -10838.756,E2 -10838.756} C_VEL
LIN {X 0,Y 404.128,Z 471.771,A -85,B 0,C 180,E1 -10841.599,E2 -10841.599} C_VEL
LIN {X 0,Y 404.15,Z 471.768,A -85,B 0,C 180,E1 -10844.521,E2 -10844.521} C_VEL
LIN {X 0,Y 404.141,Z 471.767,A -85,B 0,C 180,E1 -10847.295,E2 -10847.295} C_VEL
LIN {X 0,Y 404.173,Z 471.765,A -85,B 0,C 180,E1 -10849.955,E2 -10849.955} C_VEL
LIN {X 0,Y 404.14,Z 471.769,A -85,B 0,C 180,E1 -10853.124,E2 -10853.124} C_VEL
LIN {X 0,Y 404.149,Z 471.768,A -85,B 0,C 180,E1 -10856.187,E2 -10856.187} C_VEL
LIN {X 0,Y 404.139,Z 471.818,A -85,B 0,C 180,E1 -10857.792,E2 -10857.792} C_VEL
LIN {X 0,Y 407.937,Z 486.146,A -85,B 0,C 180,E1 -10860.592,E2 -10860.592} C_VEL
LIN {X 0,Y 410.795,Z 498.227,A -85,B 0,C 180,E1 -10862.827,E2 -10862.827} C_VEL
LIN {X 0,Y 410.771,Z 501.657,A -85,B 0,C 180,E1 -10863.392,E2 -10863.392} C_VEL
LIN {X 0,Y 408.781,Z 522.661,A -85,B 0,C 180,E1 -10866.706,E2 -10866.706} C_VEL
LIN {X 0,Y 412.57,Z 548.4,A -85,B 0,C 180,E1 -10867.41,E2 -10867.41} C_VEL
LIN {X 0,Y 410.737,Z 654.046,A -85,B 0,C 180,E1 -10869.399,E2 -10869.399} C_VEL
LIN {X 0,Y 410.192,Z 667.829,A -85,B 0,C 180,E1 -10869.796,E2 -10869.796} C_VEL
LIN {X 0,Y 409.394,Z 681.475,A -85,B 0,C 180,E1 -10870.376,E2 -10870.376} C_VEL
LIN {X 0,Y 408.519,Z 695.484,A -85,B 0,C 180,E1 -10871.196,E2 -10871.196} C_VEL
LIN {X 0,Y 407.662,Z 708.407,A -85,B 0,C 180,E1 -10872.18,E2 -10872.18} C_VEL
LIN {X 0,Y 406.58,Z 720.316,A -85,B 0,C 180,E1 -10873.298,E2 -10873.298} C_VEL
LIN {X 0,Y 405.566,Z 732.22,A -85,B 0,C 180,E1 -10874.676,E2 -10874.676} C_VEL
LIN {X 0,Y 404.737,Z 742.755,A -85,B 0,C 180,E1 -10876.169,E2 -10876.169} C_VEL
LIN {X 0,Y 404.127,Z 751.623,A -85,B 0,C 180,E1 -10877.699,E2 -10877.699} C_VEL
LIN {X 0,Y 403.547,Z 759.966,A -85,B 0,C 180,E1 -10879.462,E2 -10879.462} C_VEL
LIN {X 0,Y 403.243,Z 765.835,A -85,B 0,C 180,E1 -10880.974,E2 -10880.974} C_VEL
LIN {X 0,Y 403.056,Z 771.962,A -85,B 0,C 180,E1 -10882.988,E2 -10882.988} C_VEL
LIN {X 0,Y 402.986,Z 776.426,A -85,B 0,C 180,E1 -10884.996,E2 -10884.996} C_VEL
LIN {X 0,Y 402.965,Z 779.353,A -85,B 0,C 180,E1 -10887,E2 -10887} C_VEL
LIN {X 0,Y 402.989,Z 780.267,A -85,B 0,C 180,E1 -10888,E2 -10888} C_VEL
LIN {X 0,Y 402.939,Z 780.998,A -85,B 0,C 180,E1 -10889.999,E2 -10889.999} C_VEL
LIN {X 0,Y 402.989,Z 780.267,A -85,B 0,C 180,E1 -10891.998,E2 -10891.998} C_VEL
LIN {X 0,Y 402.9,Z 778.073,A -85,B 0,C 180,E1 -10894,E2 -10894} C_VEL
LIN {X 0,Y 402.968,Z 775.484,A -85,B 0,C 180,E1 -10895.503,E2 -10895.503} C_VEL
LIN {X 0,Y 403.054,Z 770.596,A -85,B 0,C 180,E1 -10897.513,E2 -10897.513} C_VEL
LIN {X 0,Y 403.24,Z 765.827,A -85,B 0,C 180,E1 -10899.023,E2 -10899.023} C_VEL
LIN {X 0,Y 403.613,Z 758.895,A -85,B 0,C 180,E1 -10900.787,E2 -10900.787} C_VEL
LIN {X 0,Y 404.101,Z 751.609,A -85,B 0,C 180,E1 -10902.3,E2 -10902.3} C_VEL
LIN {X 0,Y 404.736,Z 742.798,A -85,B 0,C 180,E1 -10903.819,E2 -10903.819} C_VEL
LIN {X 0,Y 405.548,Z 732.196,A -85,B 0,C 180,E1 -10905.322,E2 -10905.322} C_VEL
LIN {X 0,Y 406.467,Z 721.481,A -85,B 0,C 180,E1 -10906.575,E2 -10906.575} C_VEL
LIN {X 0,Y 407.445,Z 709.81,A -85,B 0,C 180,E1 -10907.697,E2 -10907.697} C_VEL
LIN {X 0,Y 408.405,Z 696.765,A -85,B 0,C 180,E1 -10908.709,E2 -10908.709} C_VEL
LIN {X 0,Y 409.326,Z 682.636,A -85,B 0,C 180,E1 -10909.559,E2 -10909.559} C_VEL
LIN {X 0,Y 410.115,Z 668.607,A -85,B 0,C 180,E1 -10910.173,E2 -10910.173} C_VEL
LIN {X 0,Y 410.755,Z 653.885,A -85,B 0,C 180,E1 -10910.597,E2 -10910.597} C_VEL
LIN {X 0,Y 412.504,Z 547.751,A -85,B 0,C 180,E1 -10912.597,E2 -10912.597} C_VEL
LIN {X 0,Y 408.761,Z 522.391,A -85,B 0,C 180,E1 -10913.292,E2 -10913.292} C_VEL
LIN {X 0,Y 410.847,Z 500.458,A -85,B 0,C 180,E1 -10916.791,E2 -10916.791} C_VEL
LIN {X 0,Y 410.543,Z 497.188,A -85,B 0,C 180,E1 -10917.351,E2 -10917.351} C_VEL
LIN {X 0,Y 407.092,Z 482.765,A -85,B 0,C 180,E1 -10920.041,E2 -10920.041} C_VEL
LIN {X 0,Y 404.143,Z 471.771,A -85,B 0,C 180,E1 -10922.239,E2 -10922.239} C_VEL
LIN {X 0,Y 404.176,Z 471.745,A -85,B 0,C 180,E1 -10925.189,E2 -10925.189} C_VEL
LIN {X 0,Y 404.158,Z 471.763,A -85,B 0,C 180,E1 -10928.754,E2 -10928.754} C_VEL
LIN {X 0,Y 404.184,Z 471.762,A -85,B 0,C 180,E1 -10931.61,E2 -10931.61} C_VEL
LIN {X 0,Y 404.19,Z 471.763,A -85,B 0,C 180,E1 -10934.528,E2 -10934.528} C_VEL
LIN {X 0,Y 404.203,Z 471.756,A -85,B 0,C 180,E1 -10937.304,E2 -10937.304} C_VEL
LIN {X 0,Y 404.16,Z 471.761,A -85,B 0,C 180,E1 -10939.954,E2 -10939.954} C_VEL
LIN {X 0,Y 404.132,Z 471.754,A -85,B 0,C 180,E1 -10943.123,E2 -10943.123} C_VEL
LIN {X 0,Y 404.135,Z 471.761,A -85,B 0,C 180,E1 -10946.187,E2 -10946.187} C_VEL
LIN {X 0,Y 404.146,Z 471.763,A -85,B 0,C 180,E1 -10949.715,E2 -10949.715} C_VEL
LIN {X 0,Y 404.185,Z 471.762,A -85,B 0,C 180,E1 -10953.122,E2 -10953.122} C_VEL
LIN {X 0,Y 404.166,Z 471.759,A -85,B 0,C 180,E1 -10955.334,E2 -10955.334} C_VEL
LIN {X 0,Y 404.127,Z 471.747,A -85,B 0,C 180,E1 -10958.58,E2 -10958.58} C_VEL
LIN {X 0,Y 404.199,Z 471.758,A -85,B 0,C 180,E1 -10961.762,E2 -10961.762} C_VEL
LIN {X 0,Y 404.197,Z 471.759,A -85,B 0,C 180,E1 -10964.882,E2 -10964.882} C_VEL
LIN {X 0,Y 404.261,Z 471.75,A -85,B 0,C 180,E1 -10967.959,E2 -10967.959} C_VEL
LIN {X 0,Y 404.421,Z 471.732,A -85,B 0,C 180,E1 -10972.099,E2 -10972.099} C_VEL
LIN {X 0,Y 404.414,Z 471.724,A -85,B 0,C 180,E1 -10974.015,E2 -10974.015} C_VEL
LIN {X 0,Y 404.472,Z 471.722,A -85,B 0,C 180,E1 -10978.009,E2 -10978.009} C_VEL
LIN {X 0,Y 404.602,Z 471.707,A -85,B 0,C 180,E1 -10980,E2 -10980} C_VEL
LIN {X 0,Y 404.413,Z 471.725,A -85,B 0,C 180,E1 -10982.989,E2 -10982.989} C_VEL
LIN {X 0,Y 404.4,Z 471.732,A -85,B 0,C 180,E1 -10986.988,E2 -10986.988} C_VEL
LIN {X 0,Y 404.26,Z 471.75,A -85,B 0,C 180,E1 -10990.012,E2 -10990.012} C_VEL
LIN {X 0,Y 404.255,Z 471.746,A -85,B 0,C 180,E1 -10993.212,E2 -10993.212} C_VEL
LIN {X 0,Y 404.208,Z 471.754,A -85,B 0,C 180,E1 -10997.009,E2 -10997.009} C_VEL
LIN {X 0,Y 404.176,Z 471.766,A -85,B 0,C 180,E1 -11000.351,E2 -11000.351} C_VEL
LIN {X 0,Y 404.159,Z 471.762,A -85,B 0,C 180,E1 -11003.575,E2 -11003.575} C_VEL
LIN {X 0,Y 404.174,Z 471.76,A -85,B 0,C 180,E1 -11005.767,E2 -11005.767} C_VEL
LIN {X 0,Y 404.189,Z 471.76,A -85,B 0,C 180,E1 -11008,E2 -11008} C_VEL
LIN {X 0,Y 404.138,Z 471.765,A -85,B 0,C 180,E1 -11011.561,E2 -11011.561} C_VEL
LIN {X 0,Y 404.177,Z 471.763,A -85,B 0,C 180,E1 -11015.017,E2 -11015.017} C_VEL
LIN {X 0,Y 404.157,Z 471.768,A -85,B 0,C 180,E1 -11018.757,E2 -11018.757} C_VEL
LIN {X 0,Y 404.142,Z 471.767,A -85,B 0,C 180,E1 -11021.605,E2 -11021.605} C_VEL
LIN {X 0,Y 404.146,Z 471.772,A -85,B 0,C 180,E1 -11024.525,E2 -11024.525} C_VEL
LIN {X 0,Y 404.205,Z 471.759,A -85,B 0,C 180,E1 -11027.307,E2 -11027.307} C_VEL
LIN {X 0,Y 404.164,Z 471.766,A -85,B 0,C 180,E1 -11029.957,E2 -11029.957} C_VEL
LIN {X 0,Y 404.136,Z 471.76,A -85,B 0,C 180,E1 -11033.126,E2 -11033.126} C_VEL
LIN {X 0,Y 404.142,Z 471.763,A -85,B 0,C 180,E1 -11036.189,E2 -11036.189} C_VEL
LIN {X 0,Y 404.152,Z 471.769,A -85,B 0,C 180,E1 -11039.717,E2 -11039.717} C_VEL
LIN {X 0,Y 404.203,Z 471.973,A -85,B 0,C 180,E1 -11040.248,E2 -11040.248} C_VEL
LIN {X 0,Y 407.059,Z 483.812,A -85,B 0,C 180,E1 -11043.052,E2 -11043.052} C_VEL
LIN {X 0,Y 408.934,Z 494.148,A -85,B 0,C 180,E1 -11045.371,E2 -11045.371} C_VEL
LIN {X 0,Y 407.886,Z 507.368,A -85,B 0,C 180,E1 -11048.019,E2 -11048.019} C_VEL
LIN {X 0,Y 407.224,Z 516.296,A -85,B 0,C 180,E1 -11049.777,E2 -11049.777} C_VEL
LIN {X 0,Y 411.862,Z 540.494,A -85,B 0,C 180,E1 -11050.456,E2 -11050.456} C_VEL
LIN {X 0,Y 410.932,Z 629.375,A -85,B 0,C 180,E1 -11051.911,E2 -11051.911} C_VEL
LIN {X 0,Y 410.521,Z 642.935,A -85,B 0,C 180,E1 -11052.343,E2 -11052.343} C_VEL
LIN {X 0,Y 409.897,Z 655.165,A -85,B 0,C 180,E1 -11052.927,E2 -11052.927} C_VEL
LIN {X 0,Y 409.243,Z 666.606,A -85,B 0,C 180,E1 -11053.669,E2 -11053.669} C_VEL
LIN {X 0,Y 408.461,Z 676.48,A -85,B 0,C 180,E1 -11054.482,E2 -11054.482} C_VEL
LIN {X 0,Y 407.611,Z 686.671,A -85,B 0,C 180,E1 -11055.524,E2 -11055.524} C_VEL
LIN {X 0,Y 406.615,Z 696.449,A -85,B 0,C 180,E1 -11056.762,E2 -11056.762} C_VEL
LIN {X 0,Y 405.651,Z 705.911,A -85,B 0,C 180,E1 -11058.256,E2 -11058.256} C_VEL
LIN {X 0,Y 404.944,Z 713.512,A -85,B 0,C 180,E1 -11059.754,E2 -11059.754} C_VEL
LIN {X 0,Y 404.313,Z 718.676,A -85,B 0,C 180,E1 -11061.001,E2 -11061.001} C_VEL
LIN {X 0,Y 403.835,Z 723.746,A -85,B 0,C 180,E1 -11062.502,E2 -11062.502} C_VEL
LIN {X 0,Y 403.466,Z 727.716,A -85,B 0,C 180,E1 -11064.002,E2 -11064.002} C_VEL
LIN {X 0,Y 403.277,Z 729.836,A -85,B 0,C 180,E1 -11065.002,E2 -11065.002} C_VEL
LIN {X 0,Y 403.301,Z 731.51,A -85,B 0,C 180,E1 -11066.004,E2 -11066.004} C_VEL
LIN {X 0,Y 403.081,Z 733.422,A -85,B 0,C 180,E1 -11067.684,E2 -11067.684} C_VEL
LIN {X 0,Y 402.345,Z 734.118,A -85,B 0,C 180,E1 -11068.513,E2 -11068.513} C_VEL
LIN {X 0,Y 399.435,Z 734.795,A -85,B 0,C 180,E1 -11069.865,E2 -11069.865} C_VEL
LIN {X 0,Y 397.038,Z 734.787,A -85,B 0,C 180,E1 -11070.958,E2 -11070.958} C_VEL
LIN {X 0,Y 396.049,Z 734.376,A -85,B 0,C 180,E1 -11071.801,E2 -11071.801} C_VEL
LIN {X 0,Y 395.988,Z 734.15,A -85,B 0,C 180,E1 -11072.085,E2 -11072.085} C_VEL
LIN {X 0,Y 396.191,Z 732.047,A -85,B 0,C 180,E1 -11074.07,E2 -11074.07} C_VEL
LIN {X 0,Y 396.276,Z 729.425,A -85,B 0,C 180,E1 -11075.599,E2 -11075.599} C_VEL
LIN {X 0,Y 396.686,Z 725.689,A -85,B 0,C 180,E1 -11077.186,E2 -11077.186} C_VEL
LIN {X 0,Y 397.101,Z 721.237,A -85,B 0,C 180,E1 -11078.653,E2 -11078.653} C_VEL
LIN {X 0,Y 397.895,Z 714.354,A -85,B 0,C 180,E1 -11080.432,E2 -11080.432} C_VEL
LIN {X 0,Y 398.703,Z 706.892,A -85,B 0,C 180,E1 -11081.955,E2 -11081.955} C_VEL
LIN {X 0,Y 399.437,Z 699.296,A -85,B 0,C 180,E1 -11083.224,E2 -11083.224} C_VEL
LIN {X 0,Y 400.581,Z 688.982,A -85,B 0,C 180,E1 -11084.609,E2 -11084.609} C_VEL
LIN {X 0,Y 401.508,Z 678.376,A -85,B 0,C 180,E1 -11085.756,E2 -11085.756} C_VEL
LIN {X 0,Y 402.483,Z 666.735,A -85,B 0,C 180,E1 -11086.746,E2 -11086.746} C_VEL
LIN {X 0,Y 403.282,Z 655.236,A -85,B 0,C 180,E1 -11087.496,E2 -11087.496} C_VEL
LIN {X 0,Y 403.888,Z 642.155,A -85,B 0,C 180,E1 -11088.123,E2 -11088.123} C_VEL
LIN {X 0,Y 404.361,Z 629.192,A -85,B 0,C 180,E1 -11088.527,E2 -11088.527} C_VEL
LIN {X 0,Y 405.219,Z 540.676,A -85,B 0,C 180,E1 -11090.003,E2 -11090.003} C_VEL
LIN {X 0,Y 400.43,Z 516.36,A -85,B 0,C 180,E1 -11090.711,E2 -11090.711} C_VEL
LIN {X 0,Y 401.623,Z 501.283,A -85,B 0,C 180,E1 -11093.734,E2 -11093.734} C_VEL
LIN {X 0,Y 402.047,Z 494.795,A -85,B 0,C 180,E1 -11095.082,E2 -11095.082} C_VEL
LIN {X 0,Y 399.651,Z 483.178,A -85,B 0,C 180,E1 -11097.768,E2 -11097.768} C_VEL
LIN {X 0,Y 397.126,Z 472.652,A -85,B 0,C 180,E1 -11100.329,E2 -11100.329} C_VEL
LIN {X 0,Y 397.124,Z 472.645,A -85,B 0,C 180,E1 -11103.719,E2 -11103.719} C_VEL
LIN {X 0,Y 397.103,Z 472.646,A -85,B 0,C 180,E1 -11107.21,E2 -11107.21} C_VEL
LIN {X 0,Y 397.109,Z 472.643,A -85,B 0,C 180,E1 -11110.446,E2 -11110.446} C_VEL
LIN {X 0,Y 397.11,Z 472.642,A -85,B 0,C 180,E1 -11113.649,E2 -11113.649} C_VEL
LIN {X 0,Y 397.108,Z 472.642,A -85,B 0,C 180,E1 -11116.521,E2 -11116.521} C_VEL
LIN {X 0,Y 397.119,Z 472.64,A -85,B 0,C 180,E1 -11120.423,E2 -11120.423} C_VEL
LIN {X 0,Y 397.116,Z 472.643,A -85,B 0,C 180,E1 -11124.266,E2 -11124.266} C_VEL
LIN {X 0,Y 397.121,Z 472.641,A -85,B 0,C 180,E1 -11126.727,E2 -11126.727} C_VEL
LIN {X 0,Y 397.189,Z 472.771,A -85,B 0,C 180,E1 -11130.701,E2 -11130.701} C_VEL
LIN {X 0,Y 400.549,Z 487.942,A -85,B 0,C 180,E1 -11133.49,E2 -11133.49} C_VEL
LIN {X 0,Y 401.586,Z 494.182,A -85,B 0,C 180,E1 -11134.611,E2 -11134.611} C_VEL
LIN {X 0,Y 400.569,Z 515.166,A -85,B 0,C 180,E1 -11138.109,E2 -11138.109} C_VEL
LIN {X 0,Y 399.926,Z 529.513,A -85,B 0,C 180,E1 -11140.495,E2 -11140.495} C_VEL
LIN {X 0,Y 402.861,Z 549.559,A -85,B 0,C 180,E1 -11141.084,E2 -11141.084} C_VEL
LIN {X 0,Y 400.969,Z 640.768,A -85,B 0,C 180,E1 -11143.091,E2 -11143.091} C_VEL
LIN {X 0,Y 400.645,Z 653.644,A -85,B 0,C 180,E1 -11143.569,E2 -11143.569} C_VEL
LIN {X 0,Y 400.055,Z 666.716,A -85,B 0,C 180,E1 -11144.264,E2 -11144.264} C_VEL
LIN {X 0,Y 399.474,Z 678.455,A -85,B 0,C 180,E1 -11145.09,E2 -11145.09} C_VEL
LIN {X 0,Y 398.888,Z 689.749,A -85,B 0,C 180,E1 -11146.11,E2 -11146.11} C_VEL
LIN {X 0,Y 398.233,Z 700.038,A -85,B 0,C 180,E1 -11147.256,E2 -11147.256} C_VEL
LIN {X 0,Y 397.621,Z 709.346,A -85,B 0,C 180,E1 -11148.53,E2 -11148.53} C_VEL
LIN {X 0,Y 397.057,Z 718.382,A -85,B 0,C 180,E1 -11150.062,E2 -11150.062} C_VEL
LIN {X 0,Y 396.614,Z 725.635,A -85,B 0,C 180,E1 -11151.594,E2 -11151.594} C_VEL
LIN {X 0,Y 396.277,Z 731.96,A -85,B 0,C 180,E1 -11153.303,E2 -11153.303} C_VEL
LIN {X 0,Y 396.08,Z 736.524,A -85,B 0,C 180,E1 -11154.91,E2 -11154.91} C_VEL
LIN {X 0,Y 395.952,Z 738.775,A -85,B 0,C 180,E1 -11155.929,E2 -11155.929} C_VEL
LIN {X 0,Y 395.951,Z 740.532,A -85,B 0,C 180,E1 -11156.947,E2 -11156.947} C_VEL
LIN {X 0,Y 395.918,Z 741.873,A -85,B 0,C 180,E1 -11157.965,E2 -11157.965} C_VEL
LIN {X 0,Y 395.837,Z 742.77,A -85,B 0,C 180,E1 -11158.983,E2 -11158.983} C_VEL
LIN {X 0,Y 395.82,Z 743.215,A -85,B 0,C 180,E1 -11160,E2 -11160} C_VEL
LIN {X 0,Y 395.858,Z 743.252,A -85,B 0,C 180,E1 -11161.017,E2 -11161.017} C_VEL
LIN {X 0,Y 395.938,Z 742.863,A -85,B 0,C 180,E1 -11162.034,E2 -11162.034} C_VEL
LIN {X 0,Y 396.07,Z 742.009,A -85,B 0,C 180,E1 -11163.051,E2 -11163.051} C_VEL
LIN {X 0,Y 396.159,Z 740.75,A -85,B 0,C 180,E1 -11164.069,E2 -11164.069} C_VEL
LIN {X 0,Y 396.23,Z 738.024,A -85,B 0,C 180,E1 -11165.598,E2 -11165.598} C_VEL
LIN {X 0,Y 396.592,Z 734.212,A -85,B 0,C 180,E1 -11167.126,E2 -11167.126} C_VEL
LIN {X 0,Y 396.979,Z 729.224,A -85,B 0,C 180,E1 -11168.655,E2 -11168.655} C_VEL
LIN {X 0,Y 397.594,Z 722.852,A -85,B 0,C 180,E1 -11170.181,E2 -11170.181} C_VEL
LIN {X 0,Y 398.236,Z 714.899,A -85,B 0,C 180,E1 -11171.709,E2 -11171.709} C_VEL
LIN {X 0,Y 398.901,Z 706.822,A -85,B 0,C 180,E1 -11172.981,E2 -11172.981} C_VEL
LIN {X 0,Y 399.778,Z 696.894,A -85,B 0,C 180,E1 -11174.248,E2 -11174.248} C_VEL
LIN {X 0,Y 400.676,Z 685.814,A -85,B 0,C 180,E1 -11175.385,E2 -11175.385} C_VEL
LIN {X 0,Y 401.359,Z 675.082,A -85,B 0,C 180,E1 -11176.27,E2 -11176.27} C_VEL
LIN {X 0,Y 402.146,Z 662.141,A -85,B 0,C 180,E1 -11177.087,E2 -11177.087} C_VEL
LIN {X 0,Y 402.735,Z 649.284,A -85,B 0,C 180,E1 -11177.683,E2 -11177.683} C_VEL
LIN {X 0,Y 403.232,Z 634.885,A -85,B 0,C 180,E1 -11178.12,E2 -11178.12} C_VEL
LIN {X 0,Y 405.838,Z 554.75,A -85,B 0,C 180,E1 -11180.082,E2 -11180.082} C_VEL
LIN {X 0,Y 405.944,Z 549.529,A -85,B 0,C 180,E1 -11180.222,E2 -11180.222} C_VEL
LIN {X 0,Y 403.141,Z 535.137,A -85,B 0,C 180,E1 -11180.872,E2 -11180.872} C_VEL
LIN {X 0,Y 402.593,Z 532.782,A -85,B 0,C 180,E1 -11181.002,E2 -11181.002} C_VEL
LIN {X 0,Y 403.952,Z 510.729,A -85,B 0,C 180,E1 -11184.68,E2 -11184.68} C_VEL
LIN {X 0,Y 404.602,Z 499.593,A -85,B 0,C 180,E1 -11186.569,E2 -11186.569} C_VEL
LIN {X 0,Y 403.209,Z 491.839,A -85,B 0,C 180,E1 -11188.074,E2 -11188.074} C_VEL
LIN {X 0,Y 400.491,Z 482.392,A -85,B 0,C 180,E1 -11190.075,E2 -11190.075} C_VEL
LIN {X 0,Y 397.106,Z 472.648,A -85,B 0,C 180,E1 -11192.369,E2 -11192.369} C_VEL
LIN {X 0,Y 397.114,Z 472.644,A -85,B 0,C 180,E1 -11195.734,E2 -11195.734} C_VEL
LIN {X 0,Y 397.12,Z 472.645,A -85,B 0,C 180,E1 -11199.576,E2 -11199.576} C_VEL
LIN {X 0,Y 397.107,Z 472.644,A -85,B 0,C 180,E1 -11203.478,E2 -11203.478} C_VEL
LIN {X 0,Y 397.107,Z 472.645,A -85,B 0,C 180,E1 -11206.52,E2 -11206.52} C_VEL
LIN {X 0,Y 397.117,Z 472.64,A -85,B 0,C 180,E1 -11210.422,E2 -11210.422} C_VEL
LIN {X 0,Y 397.112,Z 472.643,A -85,B 0,C 180,E1 -11214.265,E2 -11214.265} C_VEL
LIN {X 0,Y 397.117,Z 472.655,A -85,B 0,C 180,E1 -11217.331,E2 -11217.331} C_VEL
LIN {X 0,Y 401.085,Z 487.682,A -85,B 0,C 180,E1 -11220.338,E2 -11220.338} C_VEL
LIN {X 0,Y 404.109,Z 500.721,A -85,B 0,C 180,E1 -11222.795,E2 -11222.795} C_VEL
LIN {X 0,Y 402.491,Z 517.382,A -85,B 0,C 180,E1 -11225.498,E2 -11225.498} C_VEL
LIN {X 0,Y 401.997,Z 522.332,A -85,B 0,C 180,E1 -11226.306,E2 -11226.306} C_VEL
LIN {X 0,Y 405.881,Z 548.371,A -85,B 0,C 180,E1 -11227.047,E2 -11227.047} C_VEL
LIN {X 0,Y 404.288,Z 641.546,A -85,B 0,C 180,E1 -11228.822,E2 -11228.822} C_VEL
LIN {X 0,Y 403.798,Z 660.154,A -85,B 0,C 180,E1 -11229.229,E2 -11229.229} C_VEL
LIN {X 0,Y 403.115,Z 674.811,A -85,B 0,C 180,E1 -11229.758,E2 -11229.758} C_VEL
LIN {X 0,Y 402.272,Z 687.664,A -85,B 0,C 180,E1 -11230.413,E2 -11230.413} C_VEL
LIN {X 0,Y 401.339,Z 700.717,A -85,B 0,C 180,E1 -11231.285,E2 -11231.285} C_VEL
LIN {X 0,Y 400.384,Z 713.475,A -85,B 0,C 180,E1 -11232.373,E2 -11232.373} C_VEL
LIN {X 0,Y 399.306,Z 724.432,A -85,B 0,C 180,E1 -11233.511,E2 -11233.511} C_VEL
LIN {X 0,Y 398.338,Z 735.5,A -85,B 0,C 180,E1 -11234.915,E2 -11234.915} C_VEL
LIN {X 0,Y 397.514,Z 745.793,A -85,B 0,C 180,E1 -11236.506,E2 -11236.506} C_VEL
